C07163=1015.191,-31.274,-116.059,-24.116,21.567,-43.277
C07164=1015.192,-30.876,-116.091,-24.117,21.566,-43.271
C07165=1015.193,-30.478,-116.124,-24.117,21.565,-43.265
C07166=1015.195,-30.081,-116.155,-24.118,21.565,-43.260
C07167=1015.196,-29.684,-116.187,-24.119,21.565,-43.255
C07168=1015.197,-29.286,-116.220,-24.120,21.564,-43.249
C07169=1015.197,-28.889,-116.253,-24.120,21.563,-43.243
C07170=1015.198,-28.491,-116.285,-24.121,21.562,-43.238
C07171=1015.198,-28.094,-116.317,-24.122,21.562,-43.232
C07172=1015.200,-27.696,-116.350,-24.123,21.562,-43.227
C07173=1015.201,-27.299,-116.382,-24.123,21.561,-43.221
C07174=1015.201,-26.902,-116.414,-24.124,21.560,-43.217
C07175=1015.203,-26.504,-116.447,-24.125,21.560,-43.212
C07176=1015.203,-26.106,-116.479,-24.125,21.559,-43.206
C07177=1015.204,-25.709,-116.512,-24.126,21.558,-43.201
C07178=1015.205,-25.311,-116.544,-24.127,21.558,-43.195
C07179=1015.206,-24.914,-116.576,-24.128,21.558,-43.190
C07180=1015.206,-24.517,-116.610,-24.128,21.557,-43.184
C07181=1015.207,-24.120,-116.642,-24.129,21.556,-43.178
C07182=1015.207,-23.721,-116.675,-24.130,21.556,-43.173
C07183=1015.208,-23.324,-116.707,-24.131,21.555,-43.168
C07184=1015.209,-22.927,-116.740,-24.131,21.555,-43.162
C07185=1015.209,-22.529,-116.772,-24.132,21.554,-43.156
C07186=1015.210,-22.131,-116.805,-24.133,21.554,-43.151
C07187=1015.210,-21.734,-116.838,-24.134,21.553,-43.146
C07188=1015.210,-21.336,-116.870,-24.134,21.552,-43.140
C07189=1015.211,-20.939,-116.903,-24.135,21.553,-43.135
C07190=1015.212,-20.541,-116.936,-24.136,21.552,-43.129
C07191=1015.213,-20.144,-116.969,-24.136,21.551,-43.123
C07192=1015.213,-19.733,-117.002,-24.138,21.551,-43.116
C07193=1015.213,-19.483,-117.023,-24.138,21.550,-43.113
C07194=1015.213,-19.196,-117.047,-24.139,21.550,-43.109
C07195=1015.214,-18.884,-117.073,-24.139,21.550,-43.107
C07196=1015.215,-18.573,-117.098,-24.139,21.549,-43.105
C07197=1015.214,-18.285,-117.121,-24.139,21.549,-43.101
C07198=1015.214,-18.036,-117.142,-24.140,21.548,-43.098
C07199=1015.215,-17.626,-117.176,-24.141,21.547,-43.090
C07200=1015.215,-17.228,-117.209,-24.142,21.548,-43.085
C07201=1015.215,-16.831,-117.242,-24.142,21.547,-43.079
C07202=1015.216,-16.432,-117.274,-24.143,21.546,-43.074
C07203=1015.216,-16.032,-117.308,-24.144,21.546,-43.068
C07204=1015.217,-15.631,-117.341,-24.145,21.545,-43.063
C07205=1015.217,-15.228,-117.375,-24.145,21.545,-43.057
C07206=1015.216,-14.822,-117.408,-24.146,21.544,-43.052
C07207=1015.216,-14.414,-117.442,-24.147,21.544,-43.046
C07208=1015.217,-14.003,-117.476,-24.148,21.543,-43.041
C07209=1015.217,-13.588,-117.510,-24.148,21.543,-43.035
C07210=1015.217,-13.171,-117.545,-24.149,21.542,-43.029
C07211=1015.217,-12.751,-117.580,-24.150,21.542,-43.024
C07212=1015.217,-12.540,-117.598,-24.150,21.541,-43.022
C07213=1015.217,-12.329,-117.615,-24.151,21.541,-43.019
C07214=1015.217,-12.117,-117.633,-24.151,21.540,-43.016
C07215=1015.217,-11.905,-117.650,-24.151,21.540,-43.013
C07216=1015.217,-11.692,-117.668,-24.152,21.540,-43.011
C07217=1015.217,-11.479,-117.686,-24.152,21.540,-43.007
C07218=1015.217,-11.265,-117.704,-24.152,21.539,-43.006
C07219=1015.217,-11.051,-117.722,-24.153,21.539,-43.002
C07220=1015.216,-10.836,-117.740,-24.153,21.539,-42.998
C07221=1015.217,-10.621,-117.758,-24.154,21.538,-42.996
C07222=1015.216,-10.406,-117.776,-24.154,21.539,-42.993
C07223=1015.217,-10.189,-117.794,-24.154,21.538,-42.991
C07224=1015.217,-9.974,-117.811,-24.155,21.538,-42.987
C07225=1015.217,-9.758,-117.829,-24.155,21.538,-42.985
C07226=1015.216,-9.541,-117.848,-24.156,21.537,-42.982
C07227=1015.216,-9.325,-117.865,-24.156,21.537,-42.980
C07228=1015.216,-9.109,-117.883,-24.156,21.536,-42.976
C07229=1015.217,-8.892,-117.902,-24.157,21.537,-42.973
C07230=1015.217,-8.675,-117.920,-24.157,21.536,-42.971
C07231=1015.216,-8.459,-117.938,-24.158,21.536,-42.967
C07232=1015.216,-8.242,-117.956,-24.158,21.536,-42.965
C07233=1015.216,-8.026,-117.974,-24.158,21.535,-42.961
C07234=1015.216,-7.807,-117.992,-24.159,21.535,-42.959
C07235=1015.216,-7.588,-118.011,-24.159,21.534,-42.956
C07236=1015.216,-7.368,-118.029,-24.160,21.535,-42.952
C07237=1015.216,-7.146,-118.048,-24.160,21.534,-42.950
C07238=1015.216,-6.924,-118.067,-24.160,21.534,-42.947
C07239=1015.215,-6.701,-118.085,-24.161,21.533,-42.944
C07240=1015.216,-6.476,-118.104,-24.161,21.533,-42.941
C07241=1015.215,-6.252,-118.122,-24.161,21.533,-42.939
C07242=1015.215,-6.028,-118.142,-24.162,21.533,-42.935
C07243=1015.215,-5.804,-118.160,-24.162,21.532,-42.934
C07244=1015.215,-5.580,-118.179,-24.163,21.532,-42.930
C07245=1015.214,-5.357,-118.198,-24.163,21.532,-42.927
C07246=1015.214,-5.136,-118.216,-24.163,21.532,-42.925
C07247=1015.214,-4.917,-118.234,-24.164,21.531,-42.921
C07248=1015.213,-4.698,-118.253,-24.164,21.531,-42.919
C07249=1015.213,-4.481,-118.271,-24.165,21.531,-42.915
C07250=1015.213,-4.266,-118.290,-24.165,21.530,-42.913
C07251=1015.213,-4.052,-118.307,-24.165,21.530,-42.910
C07252=1015.213,-3.840,-118.325,-24.166,21.530,-42.908
C07253=1015.213,-3.629,-118.343,-24.166,21.530,-42.904
C07254=1015.212,-3.208,-118.379,-24.167,21.529,-42.899
C07255=1015.211,-2.788,-118.414,-24.168,21.529,-42.893
C07256=1015.211,-2.371,-118.449,-24.169,21.529,-42.888
C07257=1015.210,-1.955,-118.484,-24.169,21.528,-42.882
C07258=1015.210,-1.543,-118.518,-24.170,21.527,-42.877
C07259=1015.209,-1.133,-118.553,-24.171,21.527,-42.872
C07260=1015.209,-0.725,-118.588,-24.171,21.526,-42.867
C07261=1015.209,-0.320,-118.622,-24.172,21.525,-42.862
C07262=1015.208,0.084,-118.656,-24.173,21.525,-42.857
C07263=1015.207,0.486,-118.690,-24.173,21.525,-42.851
C07264=1015.206,0.885,-118.724,-24.174,21.525,-42.846
C07265=1015.206,1.284,-118.758,-24.175,21.523,-42.841
C07266=1015.206,1.682,-118.791,-24.175,21.524,-42.836
C07267=1015.205,2.068,-118.824,-24.176,21.523,-42.833
C07268=1015.203,2.420,-118.854,-24.177,21.522,-42.827
C07269=1015.203,2.744,-118.881,-24.177,21.522,-42.823
C07270=1015.203,3.056,-118.907,-24.178,21.521,-42.817
C07271=1015.202,3.384,-118.935,-24.179,21.521,-42.812
C07272=1015.202,3.744,-118.966,-24.179,21.521,-42.809
C07273=1015.200,4.133,-118.999,-24.180,21.520,-42.805
C07274=1015.199,4.529,-119.032,-24.180,21.519,-42.799
C07275=1015.199,4.924,-119.066,-24.181,21.520,-42.794
C07276=1015.198,5.319,-119.100,-24.182,21.519,-42.790
C07277=1015.197,5.714,-119.133,-24.182,21.518,-42.785
C07278=1015.196,6.108,-119.167,-24.183,21.519,-42.779
C07279=1015.195,6.500,-119.200,-24.184,21.517,-42.775
C07280=1015.194,6.893,-119.233,-24.185,21.517,-42.770
C07281=1015.193,7.284,-119.267,-24.185,21.517,-42.764
C07282=1015.193,7.671,-119.300,-24.186,21.516,-42.761
C07283=1015.191,8.055,-119.333,-24.187,21.516,-42.755
C07284=1015.190,8.436,-119.365,-24.187,21.515,-42.751
C07285=1015.190,8.815,-119.397,-24.188,21.515,-42.746
C07286=1015.189,9.191,-119.430,-24.189,21.514,-42.740
C07287=1015.187,9.566,-119.462,-24.189,21.514,-42.737
C07288=1015.186,9.943,-119.493,-24.190,21.513,-42.731
C07289=1015.185,10.321,-119.526,-24.191,21.513,-42.726
C07290=1015.184,10.702,-119.559,-24.191,21.513,-42.722
C07291=1015.183,11.085,-119.591,-24.192,21.512,-42.716
C07292=1015.182,11.470,-119.625,-24.192,21.511,-42.713
C07293=1015.181,11.856,-119.657,-24.193,21.512,-42.707
C07294=1015.179,12.244,-119.690,-24.193,21.510,-42.703
C07295=1015.178,12.630,-119.723,-24.194,21.510,-42.698
C07296=1015.177,13.016,-119.757,-24.195,21.511,-42.693
C07297=1015.176,13.403,-119.790,-24.196,21.509,-42.689
C07298=1015.175,13.791,-119.823,-24.196,21.509,-42.683
C07299=1015.173,14.178,-119.856,-24.197,21.509,-42.680
C07300=1015.172,14.566,-119.890,-24.198,21.508,-42.674
C07301=1015.171,14.955,-119.924,-24.198,21.508,-42.670
C07302=1015.169,15.345,-119.957,-24.199,21.507,-42.665
C07303=1015.168,15.735,-119.990,-24.200,21.507,-42.659
C07304=1015.166,16.126,-120.024,-24.200,21.506,-42.656
C07305=1015.165,16.517,-120.058,-24.201,21.506,-42.650
C07306=1015.163,16.910,-120.092,-24.201,21.505,-42.646
C07307=1015.162,17.304,-120.126,-24.202,21.505,-42.641
C07308=1015.161,17.698,-120.159,-24.203,21.505,-42.635
C07309=1015.159,18.094,-120.193,-24.203,21.504,-42.632
C07310=1015.158,18.489,-120.227,-24.204,21.503,-42.626
C07311=1015.156,18.886,-120.262,-24.205,21.503,-42.622
C07312=1015.155,19.282,-120.296,-24.205,21.503,-42.617
C07313=1015.154,19.493,-120.314,-24.206,21.503,-42.613
C07314=1015.153,19.730,-120.334,-24.206,21.502,-42.610
C07315=1015.151,19.995,-120.358,-24.207,21.503,-42.606
C07316=1015.151,20.282,-120.382,-24.207,21.501,-42.604
C07317=1015.149,20.579,-120.408,-24.207,21.501,-42.602
C07318=1015.148,20.871,-120.434,-24.208,21.502,-42.599
C07319=1015.147,21.143,-120.457,-24.208,21.501,-42.597
C07320=1015.146,21.387,-120.478,-24.209,21.501,-42.593
C07321=1015.145,21.802,-120.514,-24.210,21.501,-42.586
C07322=1015.143,22.176,-120.546,-24.210,21.500,-42.584
C07323=1015.142,22.498,-120.574,-24.211,21.500,-42.580
C07324=1015.140,22.764,-120.598,-24.211,21.500,-42.577
C07325=1015.139,22.996,-120.617,-24.211,21.499,-42.573
C07326=1015.138,23.230,-120.637,-24.212,21.498,-42.567
C07327=1015.137,23.502,-120.661,-24.213,21.498,-42.564
C07328=1015.135,23.832,-120.690,-24.213,21.498,-42.562
C07329=1015.134,24.215,-120.723,-24.213,21.497,-42.558
C07330=1015.132,24.614,-120.758,-24.214,21.497,-42.553
C07331=1015.130,25.014,-120.792,-24.215,21.497,-42.549
C07332=1015.129,25.413,-120.827,-24.215,21.496,-42.543
C07333=1015.126,25.812,-120.862,-24.216,21.496,-42.540
C07334=1015.124,26.212,-120.897,-24.217,21.496,-42.534
C07335=1015.122,26.611,-120.932,-24.218,21.495,-42.529
C07336=1015.121,27.010,-120.966,-24.218,21.494,-42.525
C07337=1015.119,27.410,-121.001,-24.219,21.495,-42.520
C07338=1015.116,27.809,-121.035,-24.219,21.493,-42.516
C07339=1015.114,28.208,-121.071,-24.220,21.493,-42.510
C07340=1015.112,28.608,-121.105,-24.221,21.493,-42.507
C07341=1015.110,29.008,-121.141,-24.221,21.492,-42.501
C07342=1015.108,29.408,-121.175,-24.222,21.492,-42.497
C07343=1015.106,29.807,-121.210,-24.223,21.492,-42.492
C07344=1015.104,30.206,-121.245,-24.223,21.491,-42.488
C07345=1015.102,30.606,-121.279,-24.224,21.491,-42.483
C07346=1015.100,31.006,-121.315,-24.224,21.490,-42.479
C07347=1015.098,31.404,-121.350,-24.225,21.490,-42.474
C07348=1015.095,31.804,-121.384,-24.226,21.489,-42.469
C07349=1015.093,32.204,-121.420,-24.226,21.489,-42.464
C07350=1015.091,32.604,-121.454,-24.227,21.489,-42.461
C07351=1015.089,33.003,-121.490,-24.228,21.489,-42.455
C07352=1015.086,33.403,-121.524,-24.228,21.487,-42.451
C07353=1015.084,33.803,-121.559,-24.229,21.488,-42.446
C07354=1015.082,34.202,-121.595,-24.229,21.487,-42.442
C07355=1015.079,34.602,-121.630,-24.230,21.486,-42.437
C07356=1015.077,35.002,-121.665,-24.231,21.486,-42.433
C07357=1015.075,35.402,-121.699,-24.231,21.486,-42.428
C07358=1015.073,35.801,-121.735,-24.232,21.486,-42.424
C07359=1015.070,36.201,-121.770,-24.233,21.485,-42.418
C07360=1015.068,36.601,-121.805,-24.233,21.484,-42.414
C07361=1015.065,37.001,-121.840,-24.234,21.485,-42.409
C07362=1015.063,37.401,-121.876,-24.235,21.484,-42.405
C07363=1015.060,37.801,-121.910,-24.235,21.483,-42.400
C07364=1015.058,38.200,-121.946,-24.236,21.483,-42.396
C07365=1015.055,38.600,-121.981,-24.237,21.483,-42.391
C07366=1015.053,39.000,-122.016,-24.237,21.483,-42.387
C07367=1015.050,39.400,-122.051,-24.238,21.482,-42.383
C07368=1015.047,39.800,-122.087,-24.238,21.481,-42.378
C07369=1015.045,40.200,-122.122,-24.239,21.481,-42.374
C07370=1015.042,40.600,-122.158,-24.240,21.481,-42.369
C07371=1015.040,41.000,-122.192,-24.240,21.481,-42.365
C07372=1015.037,41.399,-122.228,-24.241,21.480,-42.359
C07373=1015.033,41.799,-122.263,-24.241,21.479,-42.356
C07374=1015.031,42.199,-122.298,-24.242,21.479,-42.352
C07375=1015.028,42.599,-122.333,-24.243,21.479,-42.347
C07376=1015.025,42.999,-122.369,-24.243,21.479,-42.343
C07377=1015.023,43.399,-122.404,-24.244,21.479,-42.338
C07378=1015.020,43.799,-122.439,-24.244,21.477,-42.333
C07379=1015.017,44.199,-122.475,-24.245,21.477,-42.330
C07380=1015.014,44.599,-122.510,-24.246,21.477,-42.325
C07381=1015.011,44.999,-122.546,-24.246,21.477,-42.321
C07382=1015.009,45.399,-122.581,-24.247,21.477,-42.316
C07383=1015.006,45.799,-122.617,-24.247,21.475,-42.311
C07384=1015.003,46.199,-122.652,-24.248,21.475,-42.308
C07385=1015.000,46.599,-122.688,-24.249,21.475,-42.302
C07386=1014.997,46.999,-122.723,-24.249,21.475,-42.299
C07387=1014.994,47.400,-122.758,-24.250,21.474,-42.295
C07388=1014.991,47.799,-122.794,-24.251,21.474,-42.290
C07389=1014.987,48.200,-122.830,-24.251,21.474,-42.286
C07390=1014.985,48.599,-122.865,-24.251,21.472,-42.282
C07391=1014.982,49.000,-122.901,-24.252,21.473,-42.277
C07392=1014.979,49.400,-122.937,-24.253,21.472,-42.273
C07393=1014.975,49.800,-122.972,-24.254,21.472,-42.268
C07394=1014.973,50.200,-123.007,-24.254,21.472,-42.264
C07395=1014.970,50.600,-123.043,-24.255,21.471,-42.260
C07396=1014.966,51.001,-123.078,-24.255,21.471,-42.255
C07397=1014.963,51.401,-123.115,-24.256,21.471,-42.251
C07398=1014.960,51.801,-123.150,-24.256,21.470,-42.247
C07399=1014.957,52.201,-123.186,-24.257,21.469,-42.243
C07400=1014.953,52.601,-123.221,-24.258,21.469,-42.238
C07401=1014.949,53.001,-123.257,-24.258,21.469,-42.234
C07402=1014.946,53.401,-123.293,-24.259,21.468,-42.230
C07403=1014.943,53.801,-123.328,-24.259,21.468,-42.225
C07404=1014.940,54.201,-123.364,-24.260,21.468,-42.221
C07405=1014.937,54.602,-123.400,-24.260,21.468,-42.218
C07406=1014.933,55.002,-123.435,-24.261,21.468,-42.212
C07407=1014.930,55.402,-123.471,-24.262,21.467,-42.209
C07408=1014.927,55.803,-123.506,-24.262,21.467,-42.205
C07409=1014.923,56.202,-123.542,-24.263,21.465,-42.201
C07410=1014.920,56.602,-123.578,-24.264,21.466,-42.196
C07411=1014.916,57.002,-123.614,-24.264,21.465,-42.192
C07412=1014.913,57.403,-123.650,-24.264,21.465,-42.188
C07413=1014.909,57.803,-123.685,-24.265,21.465,-42.183
C07414=1014.906,58.203,-123.721,-24.266,21.464,-42.179
C07415=1014.901,58.603,-123.757,-24.266,21.464,-42.175
C07416=1014.898,59.003,-123.793,-24.267,21.463,-42.172
C07417=1014.895,59.403,-123.828,-24.268,21.464,-42.166
C07418=1014.891,59.804,-123.865,-24.268,21.463,-42.163
C07419=1014.887,60.203,-123.900,-24.269,21.463,-42.159
C07420=1014.884,60.603,-123.936,-24.269,21.462,-42.155
C07421=1014.880,61.004,-123.972,-24.270,21.462,-42.150
C07422=1014.877,61.405,-124.008,-24.270,21.462,-42.146
C07423=1014.872,61.804,-124.044,-24.271,21.461,-42.142
C07424=1014.869,62.204,-124.079,-24.271,21.461,-42.139
C07425=1014.865,62.624,-124.118,-24.272,21.460,-42.133
C07426=1014.862,62.877,-124.140,-24.272,21.460,-42.131
C07427=1014.860,63.145,-124.164,-24.273,21.460,-42.129
C07428=1014.858,63.395,-124.187,-24.273,21.459,-42.127
C07429=1014.856,63.612,-124.205,-24.274,21.460,-42.124
C07430=1014.854,63.819,-124.224,-24.274,21.460,-42.122
C07431=1014.852,64.036,-124.244,-24.274,21.459,-42.120
C07432=1014.849,64.266,-124.265,-24.274,21.459,-42.116
C07433=1014.848,64.502,-124.286,-24.275,21.459,-42.115
C07434=1014.845,64.738,-124.307,-24.275,21.458,-42.113
C07435=1014.842,64.968,-124.328,-24.275,21.458,-42.111
C07436=1014.840,65.188,-124.348,-24.276,21.459,-42.108
C07437=1014.838,65.402,-124.367,-24.276,21.458,-42.106
C07438=1014.834,65.810,-124.404,-24.277,21.458,-42.102
C07439=1014.830,66.207,-124.440,-24.277,21.457,-42.098
C07440=1014.827,66.608,-124.475,-24.278,21.457,-42.094
C07441=1014.822,67.010,-124.511,-24.278,21.457,-42.089
C07442=1014.818,67.414,-124.548,-24.279,21.457,-42.085
C07443=1014.814,67.818,-124.584,-24.279,21.456,-42.082
C07444=1014.810,68.224,-124.621,-24.280,21.456,-42.078
C07445=1014.806,68.632,-124.658,-24.280,21.455,-42.074
C07446=1014.801,69.040,-124.694,-24.281,21.455,-42.069
C07447=1014.796,69.451,-124.731,-24.282,21.455,-42.065
C07448=1014.793,69.861,-124.769,-24.282,21.454,-42.061
C07449=1014.788,70.273,-124.806,-24.283,21.454,-42.058
C07450=1014.784,70.684,-124.842,-24.283,21.453,-42.054
C07451=1014.780,71.095,-124.880,-24.284,21.454,-42.049
C07452=1014.775,71.505,-124.917,-24.285,21.453,-42.045
C07453=1014.771,71.918,-124.953,-24.285,21.453,-42.041
C07454=1014.767,72.332,-124.991,-24.285,21.452,-42.037
C07455=1014.762,72.746,-125.028,-24.286,21.452,-42.034
C07456=1014.758,73.164,-125.067,-24.287,21.452,-42.028
C07457=1014.753,73.584,-125.105,-24.287,21.452,-42.025
C07458=1014.751,73.796,-125.123,-24.288,21.451,-42.023
C07459=1014.749,74.008,-125.142,-24.288,21.451,-42.021
C07460=1014.746,74.221,-125.162,-24.288,21.451,-42.019
C07461=1014.744,74.434,-125.181,-24.288,21.451,-42.017
C07462=1014.741,74.647,-125.200,-24.289,21.450,-42.015
C07463=1014.738,74.861,-125.220,-24.289,21.451,-42.012
C07464=1014.736,75.074,-125.239,-24.289,21.451,-42.010
C07465=1014.734,75.286,-125.258,-24.290,21.450,-42.008
C07466=1014.729,75.706,-125.296,-24.290,21.450,-42.004
C07467=1014.724,76.118,-125.333,-24.291,21.449,-42.001
C07468=1014.719,76.520,-125.370,-24.291,21.449,-41.997
C07469=1014.715,76.915,-125.405,-24.292,21.449,-41.994
C07470=1014.711,77.303,-125.441,-24.292,21.448,-41.989
C07471=1014.707,77.689,-125.476,-24.293,21.447,-41.986
C07472=1014.702,78.075,-125.511,-24.293,21.448,-41.980
C07473=1014.698,78.465,-125.546,-24.294,21.447,-41.977
C07474=1014.692,78.863,-125.582,-24.294,21.447,-41.973
C07475=1014.688,79.268,-125.618,-24.295,21.447,-41.970
C07476=1014.683,79.683,-125.656,-24.296,21.447,-41.966
C07477=1014.681,79.893,-125.675,-24.296,21.446,-41.964
C07478=1014.678,80.104,-125.694,-24.296,21.446,-41.962
C07479=1014.675,80.317,-125.713,-24.296,21.446,-41.960
C07480=1014.673,80.530,-125.733,-24.297,21.446,-41.958
C07481=1014.670,80.743,-125.752,-24.297,21.445,-41.956
C07482=1014.668,80.955,-125.772,-24.297,21.445,-41.955
C07483=1014.665,81.168,-125.791,-24.297,21.445,-41.953
C07484=1014.663,81.380,-125.810,-24.298,21.445,-41.951
C07485=1014.660,81.593,-125.829,-24.298,21.445,-41.949
C07486=1014.657,81.804,-125.848,-24.298,21.444,-41.947
C07487=1014.655,82.016,-125.867,-24.299,21.445,-41.944
C07488=1014.652,82.227,-125.887,-24.299,21.444,-41.942
C07489=1014.647,82.647,-125.924,-24.299,21.444,-41.938
C07490=1014.641,83.068,-125.963,-24.300,21.444,-41.935
C07491=1014.637,83.486,-126.001,-24.300,21.444,-41.931
C07492=1014.632,83.904,-126.039,-24.301,21.443,-41.927
C07493=1014.626,84.320,-126.077,-24.301,21.443,-41.923
C07494=1014.621,84.734,-126.115,-24.302,21.443,-41.920
C07495=1014.616,85.146,-126.151,-24.302,21.442,-41.916
C07496=1014.611,85.557,-126.189,-24.303,21.442,-41.912
C07497=1014.605,85.965,-126.226,-24.303,21.441,-41.908
C07498=1014.601,86.373,-126.263,-24.304,21.442,-41.905
C07499=1014.595,86.779,-126.300,-24.304,21.441,-41.901
C07500=1014.590,87.182,-126.336,-24.305,21.441,-41.898
C07501=1014.584,87.578,-126.373,-24.305,21.440,-41.894
C07502=1014.579,87.966,-126.408,-24.306,21.440,-41.890
C07503=1014.575,88.349,-126.443,-24.307,21.440,-41.887
C07504=1014.570,88.732,-126.477,-24.307,21.440,-41.883
C07505=1014.565,89.118,-126.513,-24.308,21.439,-41.879
C07506=1014.559,89.510,-126.548,-24.308,21.439,-41.875
C07507=1014.554,89.910,-126.585,-24.309,21.439,-41.872
C07508=1014.549,90.308,-126.621,-24.309,21.439,-41.868
C07509=1014.543,90.707,-126.658,-24.310,21.438,-41.865
C07510=1014.538,91.106,-126.693,-24.310,21.438,-41.861
C07511=1014.532,91.505,-126.730,-24.311,21.438,-41.857
C07512=1014.526,91.904,-126.767,-24.311,21.438,-41.854
C07513=1014.521,92.303,-126.803,-24.312,21.437,-41.850
C07514=1014.516,92.702,-126.839,-24.312,21.437,-41.846
C07515=1014.510,93.102,-126.875,-24.312,21.437,-41.844
C07516=1014.505,93.500,-126.911,-24.313,21.436,-41.841
C07517=1014.499,93.899,-126.948,-24.313,21.436,-41.837
C07518=1014.493,94.298,-126.984,-24.314,21.435,-41.833
C07519=1014.488,94.697,-127.020,-24.315,21.436,-41.830
C07520=1014.482,95.096,-127.057,-24.315,21.435,-41.826
C07521=1014.476,95.495,-127.093,-24.316,21.435,-41.822
C07522=1014.470,95.894,-127.130,-24.316,21.435,-41.819
C07523=1014.465,96.293,-127.166,-24.317,21.435,-41.815
C07524=1014.460,96.691,-127.202,-24.317,21.434,-41.811
C07525=1014.453,97.090,-127.238,-24.318,21.434,-41.808
C07526=1014.447,97.489,-127.275,-24.318,21.433,-41.806
C07527=1014.442,97.888,-127.311,-24.318,21.433,-41.802
C07528=1014.435,98.286,-127.348,-24.319,21.432,-41.798
C07529=1014.430,98.685,-127.384,-24.319,21.433,-41.795
C07530=1014.423,99.084,-127.420,-24.320,21.432,-41.791
C07531=1014.418,99.482,-127.456,-24.320,21.432,-41.787
C07532=1014.413,99.881,-127.493,-24.321,21.432,-41.784
C07533=1014.406,100.280,-127.529,-24.322,21.432,-41.780
C07534=1014.400,100.678,-127.565,-24.322,21.431,-41.778
C07535=1014.394,101.077,-127.602,-24.322,21.431,-41.775
C07536=1014.388,101.476,-127.638,-24.323,21.431,-41.771
C07537=1014.382,101.875,-127.675,-24.323,21.430,-41.767
C07538=1014.376,102.273,-127.711,-24.324,21.430,-41.763
C07539=1014.369,102.671,-127.747,-24.324,21.430,-41.760
C07540=1014.363,103.071,-127.784,-24.325,21.430,-41.756
C07541=1014.357,103.469,-127.821,-24.325,21.430,-41.754
C07542=1014.350,103.867,-127.857,-24.326,21.429,-41.751
C07543=1014.344,104.266,-127.893,-24.326,21.429,-41.747
C07544=1014.338,104.665,-127.930,-24.327,21.429,-41.743
C07545=1014.332,105.063,-127.966,-24.327,21.429,-41.740
C07546=1014.325,105.461,-128.002,-24.328,21.428,-41.736
C07547=1014.319,105.860,-128.038,-24.328,21.428,-41.734
C07548=1014.313,106.259,-128.075,-24.328,21.427,-41.730
C07549=1014.306,106.658,-128.112,-24.329,21.427,-41.727
C07550=1014.300,107.056,-128.148,-24.330,21.427,-41.723
C07551=1014.294,107.454,-128.184,-24.330,21.427,-41.719
C07552=1014.286,107.853,-128.221,-24.330,21.426,-41.717
C07553=1014.280,108.251,-128.257,-24.331,21.426,-41.714
C07554=1014.274,108.650,-128.293,-24.331,21.426,-41.710
C07555=1014.267,109.048,-128.330,-24.332,21.426,-41.707
C07556=1014.260,109.447,-128.366,-24.332,21.426,-41.703
C07557=1014.254,109.845,-128.402,-24.333,21.425,-41.701
C07558=1014.247,110.244,-128.439,-24.333,21.425,-41.697
C07559=1014.241,110.642,-128.475,-24.334,21.425,-41.694
C07560=1014.233,111.040,-128.512,-24.334,21.425,-41.690
C07561=1014.227,111.438,-128.548,-24.334,21.424,-41.688
C07562=1014.220,111.837,-128.585,-24.335,21.423,-41.684
C07563=1014.213,112.235,-128.621,-24.335,21.424,-41.681
C07564=1014.206,112.634,-128.658,-24.336,21.423,-41.677
C07565=1014.199,113.031,-128.694,-24.336,21.423,-41.675
C07566=1014.192,113.430,-128.731,-24.337,21.423,-41.671
C07567=1014.186,113.828,-128.767,-24.337,21.422,-41.668
C07568=1014.178,114.228,-128.803,-24.338,21.423,-41.664
C07569=1014.171,114.625,-128.839,-24.338,21.422,-41.662
C07570=1014.164,115.024,-128.876,-24.339,21.422,-41.659
C07571=1014.157,115.422,-128.912,-24.339,21.422,-41.655
C07572=1014.150,115.820,-128.948,-24.340,21.422,-41.652
C07573=1014.143,116.219,-128.985,-24.340,21.421,-41.649
C07574=1014.136,116.617,-129.021,-24.340,21.420,-41.646
C07575=1014.128,117.016,-129.058,-24.341,21.421,-41.642
C07576=1014.121,117.414,-129.093,-24.341,21.420,-41.638
C07577=1014.114,117.813,-129.130,-24.342,21.420,-41.637
C07578=1014.106,118.210,-129.167,-24.342,21.420,-41.633
C07579=1014.099,118.609,-129.203,-24.343,21.420,-41.629
C07580=1014.092,119.007,-129.240,-24.343,21.420,-41.626
C07581=1014.085,119.406,-129.275,-24.343,21.419,-41.624
C07582=1014.077,119.804,-129.312,-24.344,21.419,-41.620
C07583=1014.070,120.202,-129.348,-24.345,21.419,-41.617
C07584=1014.063,120.601,-129.385,-24.345,21.418,-41.614
C07585=1014.056,120.999,-129.422,-24.345,21.418,-41.611
C07586=1014.048,121.397,-129.458,-24.346,21.418,-41.607
C07587=1014.042,121.796,-129.494,-24.346,21.417,-41.605
C07588=1014.034,122.194,-129.531,-24.347,21.418,-41.602
C07589=1014.027,122.593,-129.568,-24.347,21.417,-41.598
C07590=1014.020,122.991,-129.605,-24.348,21.418,-41.595
C07591=1014.013,123.389,-129.641,-24.348,21.416,-41.592
C07592=1014.006,123.788,-129.678,-24.348,21.417,-41.589
C07593=1013.998,124.187,-129.715,-24.349,21.416,-41.585
C07594=1013.991,124.585,-129.751,-24.349,21.416,-41.583
C07595=1013.984,124.983,-129.788,-24.350,21.416,-41.580
C07596=1013.976,125.381,-129.825,-24.350,21.416,-41.576
C07597=1013.969,125.780,-129.861,-24.350,21.415,-41.574
C07598=1013.962,126.179,-129.898,-24.351,21.415,-41.571
C07599=1013.954,126.577,-129.935,-24.351,21.415,-41.567
C07600=1013.947,126.975,-129.971,-24.352,21.415,-41.565
C07601=1013.939,127.373,-130.008,-24.352,21.414,-41.561
C07602=1013.932,127.772,-130.045,-24.353,21.415,-41.558
C07603=1013.924,128.170,-130.082,-24.353,21.414,-41.555
C07604=1013.917,128.569,-130.119,-24.354,21.414,-41.552
C07605=1013.909,128.967,-130.155,-24.354,21.413,-41.550
C07606=1013.902,129.365,-130.192,-24.354,21.413,-41.547
C07607=1013.894,129.764,-130.228,-24.355,21.413,-41.543
C07608=1013.886,130.163,-130.265,-24.355,21.413,-41.541
C07609=1013.879,130.561,-130.301,-24.356,21.413,-41.538
C07610=1013.871,130.959,-130.338,-24.356,21.413,-41.534
C07611=1013.863,131.358,-130.375,-24.356,21.412,-41.532
C07612=1013.855,131.756,-130.411,-24.357,21.412,-41.528
C07613=1013.847,132.155,-130.448,-24.357,21.412,-41.525
C07614=1013.840,132.553,-130.485,-24.358,21.411,-41.523
C07615=1013.831,132.952,-130.522,-24.358,21.412,-41.519
C07616=1013.823,133.350,-130.558,-24.358,21.411,-41.517
C07617=1013.815,133.749,-130.595,-24.359,21.411,-41.514
C07618=1013.807,134.148,-130.631,-24.359,21.411,-41.510
C07619=1013.799,134.546,-130.668,-24.360,21.410,-41.508
C07620=1013.791,134.944,-130.704,-24.360,21.411,-41.505
C07621=1013.783,135.340,-130.741,-24.360,21.410,-41.502
C07622=1013.775,135.711,-130.774,-24.361,21.409,-41.500
C07623=1013.768,136.050,-130.806,-24.361,21.410,-41.497
C07624=1013.762,136.368,-130.835,-24.361,21.409,-41.495
C07625=1013.755,136.685,-130.864,-24.362,21.409,-41.491
C07626=1013.748,137.021,-130.895,-24.363,21.410,-41.488
C07627=1013.741,137.390,-130.928,-24.363,21.408,-41.486
C07628=1013.732,137.791,-130.965,-24.363,21.408,-41.484
C07629=1013.728,137.996,-130.984,-24.363,21.408,-41.482
C07630=1013.723,138.213,-131.004,-24.364,21.408,-41.480
C07631=1013.718,138.451,-131.026,-24.364,21.408,-41.478
C07632=1013.712,138.710,-131.050,-24.364,21.407,-41.476
C07633=1013.707,138.988,-131.075,-24.364,21.408,-41.475
C07634=1013.700,139.275,-131.101,-24.365,21.408,-41.473
C07635=1013.694,139.563,-131.128,-24.365,21.408,-41.471
C07636=1013.688,139.840,-131.153,-24.365,21.408,-41.470
C07637=1013.683,140.099,-131.177,-24.366,21.408,-41.468
C07638=1013.678,140.334,-131.199,-24.366,21.408,-41.466
C07639=1013.668,140.751,-131.236,-24.366,21.407,-41.462
C07640=1013.660,141.156,-131.273,-24.366,21.406,-41.460
C07641=1013.651,141.561,-131.311,-24.367,21.407,-41.457
C07642=1013.642,141.967,-131.348,-24.368,21.406,-41.453
C07643=1013.633,142.373,-131.386,-24.368,21.406,-41.451
C07644=1013.624,142.782,-131.423,-24.368,21.406,-41.448
C07645=1013.615,143.191,-131.460,-24.369,21.405,-41.445
C07646=1013.605,143.599,-131.497,-24.369,21.406,-41.442
C07647=1013.597,144.009,-131.534,-24.370,21.405,-41.438
C07648=1013.587,144.420,-131.572,-24.370,21.405,-41.436
C07649=1013.578,144.832,-131.610,-24.370,21.405,-41.432
C07650=1013.568,145.243,-131.648,-24.371,21.404,-41.431
C07651=1013.559,145.655,-131.685,-24.371,21.405,-41.427
C07652=1013.549,146.068,-131.723,-24.372,21.404,-41.424
C07653=1013.542,146.377,-131.751,-24.372,21.404,-41.422
C07654=1013.515,147.591,-131.861,-24.540,22.052,-41.028
C07655=1013.508,147.860,-131.887,-24.577,22.199,-40.939
C07656=1013.502,148.138,-131.912,-24.616,22.351,-40.849
C07657=1013.494,148.423,-131.937,-24.654,22.506,-40.757
C07658=1013.488,148.714,-131.963,-24.694,22.666,-40.663
C07659=1013.481,149.010,-131.991,-24.734,22.828,-40.570
C07660=1013.474,149.309,-132.018,-24.774,22.993,-40.474
C07661=1013.467,149.610,-132.045,-24.814,23.158,-40.379
C07662=1013.460,149.909,-132.073,-24.853,23.322,-40.286
C07663=1013.454,150.206,-132.099,-24.892,23.487,-40.192
C07664=1013.447,150.497,-132.126,-24.930,23.649,-40.102
C07665=1013.440,150.783,-132.152,-24.967,23.807,-40.013
C07666=1013.433,151.062,-132.177,-25.003,23.962,-39.926
C07667=1013.427,151.333,-132.202,-25.038,24.113,-39.842
C07668=1013.421,151.596,-132.225,-25.071,24.258,-39.762
C07669=1013.415,151.850,-132.249,-25.103,24.400,-39.683
C07670=1013.409,152.099,-132.271,-25.135,24.540,-39.606
C07671=1013.404,152.343,-132.293,-25.165,24.676,-39.532
C07672=1013.398,152.585,-132.315,-25.195,24.812,-39.459
C07673=1013.392,152.826,-132.337,-25.225,24.947,-39.386
C07674=1013.387,153.067,-132.358,-25.255,25.083,-39.312
C07675=1013.381,153.308,-132.381,-25.284,25.219,-39.240
C07676=1013.375,153.550,-132.402,-25.314,25.356,-39.168
C07677=1013.370,153.791,-132.424,-25.343,25.491,-39.097
C07678=1013.365,154.032,-132.445,-25.372,25.627,-39.025
C07679=1013.359,154.272,-132.467,-25.401,25.764,-38.954
C07680=1013.353,154.513,-132.489,-25.429,25.900,-38.884
C07681=1013.348,154.753,-132.511,-25.458,26.037,-38.813
C07682=1013.342,154.992,-132.533,-25.486,26.173,-38.743
C07683=1013.337,155.232,-132.554,-25.514,26.310,-38.672
C07684=1013.331,155.472,-132.575,-25.542,26.447,-38.603
C07685=1013.326,155.711,-132.597,-25.569,26.583,-38.534
C07686=1013.320,155.950,-132.619,-25.597,26.719,-38.465
C07687=1013.315,156.190,-132.640,-25.624,26.857,-38.396
C07688=1013.310,156.429,-132.662,-25.652,26.994,-38.328
C07689=1013.303,156.668,-132.683,-25.679,27.132,-38.260
C07690=1013.295,157.070,-132.719,-25.724,27.362,-38.147
C07691=1013.287,157.384,-132.748,-25.759,27.544,-38.058
C07692=1013.282,157.622,-132.769,-25.785,27.680,-37.991
C07693=1013.276,157.859,-132.790,-25.811,27.817,-37.925
C07694=1013.271,158.096,-132.811,-25.837,27.955,-37.859
C07695=1013.265,158.331,-132.832,-25.862,28.091,-37.795
C07696=1013.260,158.566,-132.854,-25.888,28.227,-37.729
C07697=1013.254,158.801,-132.875,-25.913,28.364,-37.665
C07698=1013.249,159.037,-132.896,-25.938,28.501,-37.599
C07699=1013.243,159.273,-132.916,-25.963,28.638,-37.536
C07700=1013.239,159.507,-132.938,-25.988,28.775,-37.472
C07701=1013.232,159.739,-132.958,-26.012,28.910,-37.409
C07702=1013.230,159.972,-132.981,-26.026,28.985,-37.375
C07703=1013.229,160.206,-133.005,-26.028,28.996,-37.368
C07704=1013.228,160.445,-133.030,-26.030,29.007,-37.362
C07705=1013.227,160.696,-133.056,-26.032,29.019,-37.354
C07706=1013.226,160.958,-133.083,-26.034,29.031,-37.348
C07707=1013.224,161.235,-133.112,-26.037,29.045,-37.339
C07708=1013.223,161.528,-133.143,-26.039,29.058,-37.332
C07709=1013.221,161.831,-133.174,-26.042,29.072,-37.323
C07710=1013.220,162.137,-133.206,-26.044,29.085,-37.316
C07711=1013.218,162.429,-133.236,-26.047,29.099,-37.308
C07712=1013.217,162.736,-133.269,-26.049,29.113,-37.301
C07713=1013.216,163.030,-133.299,-26.052,29.126,-37.292
C07714=1013.215,163.293,-133.326,-26.054,29.138,-37.286
C07715=1013.213,163.531,-133.351,-26.056,29.148,-37.279
C07716=1013.212,163.751,-133.374,-26.058,29.158,-37.274
C07717=1013.211,164.086,-133.409,-26.061,29.175,-37.265
C07718=1013.210,164.360,-133.438,-26.063,29.187,-37.257
C07719=1013.209,164.678,-133.471,-26.066,29.201,-37.251
C07720=1013.207,164.981,-133.503,-26.068,29.215,-37.242
C07721=1013.206,165.216,-133.527,-26.070,29.225,-37.235
C07722=1013.206,165.451,-133.551,-26.073,29.237,-37.229
C07723=1013.204,165.687,-133.576,-26.074,29.247,-37.224
C07724=1013.203,165.923,-133.601,-26.076,29.257,-37.217
C07725=1013.202,166.158,-133.625,-26.078,29.267,-37.211
C07726=1013.202,166.393,-133.650,-26.080,29.279,-37.205
C07727=1013.201,166.629,-133.675,-26.082,29.289,-37.198
C07728=1013.199,166.864,-133.699,-26.084,29.300,-37.193
C07729=1013.198,167.100,-133.724,-26.086,29.311,-37.187
C07730=1013.197,167.335,-133.748,-26.088,29.322,-37.180
C07731=1013.196,167.571,-133.773,-26.090,29.334,-37.174
C07732=1013.195,167.806,-133.798,-26.093,29.346,-37.166
C07733=1013.194,168.042,-133.823,-26.094,29.356,-37.161
C07734=1013.193,168.278,-133.847,-26.097,29.367,-37.155
C07735=1013.193,168.513,-133.872,-26.098,29.377,-37.149
C07736=1013.191,168.749,-133.896,-26.100,29.388,-37.143
C07737=1013.190,168.984,-133.921,-26.102,29.399,-37.136
C07738=1013.189,169.220,-133.946,-26.104,29.411,-37.130
C07739=1013.189,169.455,-133.970,-26.106,29.420,-37.125
C07740=1013.187,169.690,-133.995,-26.109,29.433,-37.117
C07741=1013.186,169.926,-134.020,-26.111,29.444,-37.111
C07742=1013.185,170.162,-134.045,-26.113,29.457,-37.105
C07743=1013.184,170.398,-134.070,-26.115,29.467,-37.098
C07744=1013.183,170.633,-134.095,-26.117,29.477,-37.093
C07745=1013.183,170.868,-134.119,-26.119,29.488,-37.086
C07746=1013.181,171.104,-134.144,-26.120,29.498,-37.081
C07747=1013.180,171.340,-134.169,-26.122,29.510,-37.075
C07748=1013.179,171.575,-134.193,-26.124,29.520,-37.068
C07749=1013.179,171.811,-134.218,-26.126,29.532,-37.062
C07750=1013.178,172.047,-134.242,-26.129,29.543,-37.056
C07751=1013.177,172.282,-134.267,-26.131,29.557,-37.049
C07752=1013.176,172.517,-134.292,-26.133,29.568,-37.042
C07753=1013.174,172.753,-134.317,-26.135,29.578,-37.037
C07754=1013.174,172.989,-134.342,-26.137,29.588,-37.030
C07755=1013.173,173.225,-134.367,-26.139,29.599,-37.025
C07756=1013.171,173.460,-134.392,-26.141,29.610,-37.019
C07757=1013.171,173.695,-134.416,-26.143,29.621,-37.012
C07758=1013.170,173.932,-134.441,-26.145,29.633,-37.006
C07759=1013.169,174.167,-134.466,-26.147,29.644,-37.000
C07760=1013.168,174.402,-134.491,-26.149,29.657,-36.992
C07761=1013.167,174.638,-134.516,-26.151,29.669,-36.986
C07762=1013.166,174.874,-134.541,-26.153,29.680,-36.980
C07763=1013.165,175.110,-134.565,-26.155,29.690,-36.975
C07764=1013.164,175.345,-134.590,-26.157,29.702,-36.969
C07765=1013.163,175.581,-134.616,-26.159,29.712,-36.962
C07766=1013.163,175.817,-134.640,-26.161,29.724,-36.956
C07767=1013.162,176.052,-134.665,-26.163,29.735,-36.949
C07768=1013.161,176.288,-134.690,-26.165,29.747,-36.943
C07769=1013.160,176.524,-134.715,-26.167,29.758,-36.937
C07770=1013.159,176.759,-134.740,-26.169,29.770,-36.931
C07771=1013.158,176.995,-134.765,-26.171,29.782,-36.925
C07772=1013.156,177.231,-134.789,-26.174,29.795,-36.917
C07773=1013.156,177.466,-134.815,-26.175,29.804,-36.912
C07774=1013.155,177.702,-134.840,-26.177,29.816,-36.906
C07775=1013.154,177.938,-134.864,-26.179,29.827,-36.899
C07776=1013.153,178.174,-134.890,-26.181,29.837,-36.894
C07777=1013.152,178.409,-134.915,-26.183,29.849,-36.888
C07778=1013.152,178.645,-134.939,-26.185,29.861,-36.880
C07779=1013.151,178.880,-134.964,-26.187,29.873,-36.874
C07780=1013.150,179.116,-134.989,-26.189,29.885,-36.868
C07781=1013.149,179.352,-135.014,-26.192,29.897,-36.861
C07782=1013.148,179.587,-135.039,-26.194,29.909,-36.854
C07783=1013.147,179.823,-135.064,-26.196,29.920,-36.850
C07784=1013.146,180.059,-135.089,-26.198,29.931,-36.843
C07785=1013.145,180.295,-135.114,-26.200,29.942,-36.837
C07786=1013.144,180.531,-135.139,-26.202,29.953,-36.830
C07787=1013.143,180.766,-135.164,-26.204,29.965,-36.824
C07788=1013.142,181.002,-135.189,-26.206,29.976,-36.818
C07789=1013.141,181.238,-135.214,-26.208,29.989,-36.812
C07790=1013.140,181.473,-135.239,-26.210,30.001,-36.805
C07791=1013.140,181.710,-135.264,-26.212,30.013,-36.799
C07792=1013.138,181.945,-135.289,-26.214,30.025,-36.793
C07793=1013.138,182.181,-135.314,-26.216,30.035,-36.786
C07794=1013.137,182.416,-135.340,-26.218,30.046,-36.781
C07795=1013.136,182.653,-135.364,-26.220,30.058,-36.775
C07796=1013.135,182.888,-135.389,-26.222,30.069,-36.769
C07797=1013.135,183.124,-135.415,-26.224,30.081,-36.762
C07798=1013.133,183.359,-135.440,-26.226,30.094,-36.755
C07799=1013.133,183.596,-135.465,-26.228,30.105,-36.749
C07800=1013.132,183.831,-135.490,-26.230,30.119,-36.742
C07801=1013.131,184.067,-135.515,-26.232,30.130,-36.736
C07802=1013.130,184.302,-135.540,-26.234,30.142,-36.730
C07803=1013.130,184.538,-135.566,-26.236,30.153,-36.723
C07804=1013.128,184.774,-135.590,-26.238,30.164,-36.719
C07805=1013.128,185.010,-135.616,-26.240,30.175,-36.712
C07806=1013.127,185.245,-135.641,-26.242,30.187,-36.706
C07807=1013.126,185.481,-135.666,-26.244,30.199,-36.699
C07808=1013.125,185.717,-135.691,-26.246,30.212,-36.693
C07809=1013.124,185.953,-135.716,-26.248,30.223,-36.687
C07810=1013.123,186.188,-135.741,-26.251,30.236,-36.680
C07811=1013.123,186.424,-135.767,-26.253,30.249,-36.674
C07812=1013.122,186.660,-135.792,-26.255,30.260,-36.668
C07813=1013.121,186.895,-135.817,-26.257,30.271,-36.661
C07814=1013.120,187.132,-135.842,-26.259,30.282,-36.655
C07815=1013.119,187.367,-135.867,-26.261,30.294,-36.649
C07816=1013.119,187.603,-135.892,-26.263,30.306,-36.643
C07817=1013.118,187.839,-135.917,-26.265,30.318,-36.637
C07818=1013.117,188.075,-135.943,-26.267,30.330,-36.631
C07819=1013.116,188.311,-135.969,-26.269,30.343,-36.623
C07820=1013.115,188.547,-135.993,-26.271,30.356,-36.616
C07821=1013.114,188.783,-136.019,-26.273,30.368,-36.611
C07822=1013.113,189.018,-136.044,-26.275,30.380,-36.604
C07823=1013.113,189.254,-136.069,-26.277,30.391,-36.598
C07824=1013.112,189.490,-136.095,-26.279,30.403,-36.592
C07825=1013.111,189.725,-136.120,-26.281,30.414,-36.586
C07826=1013.111,189.961,-136.145,-26.283,30.426,-36.580
C07827=1013.110,190.197,-136.171,-26.285,30.438,-36.574
C07828=1013.109,190.433,-136.195,-26.287,30.450,-36.568
C07829=1013.108,190.669,-136.221,-26.289,30.463,-36.561
C07830=1013.108,190.905,-136.246,-26.292,30.476,-36.554
C07831=1013.107,191.140,-136.271,-26.294,30.489,-36.548
C07832=1013.106,191.376,-136.297,-26.296,30.500,-36.542
C07833=1013.105,191.612,-136.323,-26.298,30.512,-36.536
C07834=1013.104,191.848,-136.348,-26.300,30.523,-36.529
C07835=1013.104,192.084,-136.373,-26.301,30.535,-36.523
C07836=1013.103,192.320,-136.399,-26.303,30.546,-36.517
C07837=1013.103,192.556,-136.424,-26.305,30.559,-36.511
C07838=1013.102,192.791,-136.449,-26.308,30.572,-36.504
C07839=1013.101,193.027,-136.475,-26.310,30.584,-36.499
C07840=1013.100,193.263,-136.499,-26.312,30.597,-36.492
C07841=1013.099,193.499,-136.525,-26.314,30.611,-36.485
C07842=1013.099,193.735,-136.550,-26.316,30.622,-36.478
C07843=1013.097,193.971,-136.576,-26.318,30.633,-36.474
C07844=1013.097,194.207,-136.602,-26.320,30.644,-36.467
C07845=1013.096,194.442,-136.627,-26.322,30.656,-36.461
C07846=1013.095,194.678,-136.652,-26.324,30.669,-36.454
C07847=1013.095,194.914,-136.678,-26.326,30.681,-36.448
C07848=1013.095,195.150,-136.703,-26.328,30.694,-36.441
C07849=1013.093,195.385,-136.728,-26.330,30.706,-36.435
C07850=1013.093,195.621,-136.754,-26.332,30.719,-36.428
C07851=1013.092,195.857,-136.780,-26.335,30.733,-36.421
C07852=1013.091,196.093,-136.805,-26.336,30.743,-36.416
C07853=1013.091,196.329,-136.831,-26.338,30.755,-36.410
C07854=1013.090,196.565,-136.856,-26.340,30.767,-36.405
C07855=1013.090,196.800,-136.882,-26.342,30.779,-36.398
C07856=1013.089,197.036,-136.907,-26.345,30.792,-36.391
C07857=1013.089,197.272,-136.933,-26.346,30.804,-36.385
C07858=1013.088,197.508,-136.958,-26.349,30.817,-36.378
C07859=1013.086,197.743,-136.984,-26.351,30.831,-36.372
C07860=1013.086,197.979,-137.009,-26.353,30.843,-36.366
C07861=1013.085,198.226,-137.036,-26.355,30.857,-36.358
C07862=1013.084,198.618,-137.078,-26.359,30.878,-36.348
C07863=1013.083,199.009,-137.121,-26.362,30.898,-36.339
C07864=1013.083,199.250,-137.147,-26.364,30.911,-36.332
C07865=1013.082,199.479,-137.172,-26.366,30.923,-36.326
C07866=1013.081,199.712,-137.197,-26.368,30.936,-36.319
C07867=1013.081,199.953,-137.223,-26.370,30.948,-36.313
C07868=1013.080,200.207,-137.250,-26.372,30.962,-36.306
C07869=1013.079,200.462,-137.279,-26.375,30.975,-36.299
C07870=1013.079,200.701,-137.304,-26.377,30.988,-36.292
C07871=1013.078,200.923,-137.329,-26.379,31.000,-36.286
C07872=1013.077,201.140,-137.352,-26.380,31.011,-36.282
C07873=1013.076,201.556,-137.397,-26.384,31.033,-36.271
C07874=1013.076,201.762,-137.420,-26.386,31.044,-36.264
C07875=1013.076,201.981,-137.443,-26.388,31.057,-36.258
C07876=1013.078,203.216,-137.580,-26.364,31.070,-36.698
C07877=1013.079,203.464,-137.607,-26.366,31.081,-36.692
C07878=1013.081,203.709,-137.634,-26.368,31.094,-36.686
C07879=1013.083,203.954,-137.660,-26.370,31.107,-36.681
C07880=1013.084,204.199,-137.687,-26.372,31.119,-36.675
C07881=1013.086,204.442,-137.714,-26.374,31.131,-36.670
C07882=1013.088,204.686,-137.740,-26.376,31.144,-36.664
C07883=1013.089,204.930,-137.767,-26.378,31.156,-36.658
C07884=1013.090,205.174,-137.794,-26.381,31.168,-36.653
C07885=1013.093,205.418,-137.821,-26.383,31.181,-36.647
C07886=1013.094,205.661,-137.848,-26.385,31.193,-36.642
C07887=1013.096,205.905,-137.874,-26.387,31.206,-36.636
C07888=1013.097,206.148,-137.900,-26.389,31.217,-36.630
C07889=1013.099,206.391,-137.927,-26.391,31.229,-36.624
C07890=1013.101,206.634,-137.954,-26.393,31.242,-36.619
C07891=1013.102,206.877,-137.981,-26.395,31.254,-36.613
C07892=1013.104,207.119,-138.007,-26.397,31.266,-36.607
C07893=1013.106,207.363,-138.033,-26.399,31.278,-36.601
C07894=1013.108,207.604,-138.060,-26.401,31.291,-36.596
C07895=1013.108,207.847,-138.087,-26.403,31.303,-36.590
C07896=1013.110,208.090,-138.113,-26.405,31.315,-36.584
C07897=1013.112,208.332,-138.140,-26.407,31.327,-36.578
C07898=1013.114,208.575,-138.166,-26.409,31.339,-36.573
C07899=1013.116,208.817,-138.193,-26.410,31.351,-36.567
C07900=1013.117,209.060,-138.220,-26.413,31.363,-36.561
C07901=1013.119,209.301,-138.246,-26.415,31.376,-36.555
C07902=1013.121,209.543,-138.273,-26.416,31.387,-36.549
C07903=1013.122,209.787,-138.300,-26.418,31.400,-36.544
C07904=1013.124,210.028,-138.327,-26.420,31.411,-36.540
C07905=1013.126,210.271,-138.353,-26.422,31.424,-36.532
C07906=1013.128,210.513,-138.380,-26.424,31.436,-36.526
C07907=1013.129,210.756,-138.407,-26.426,31.449,-36.521
C07908=1013.132,210.998,-138.434,-26.428,31.461,-36.515
C07909=1013.132,211.241,-138.460,-26.430,31.472,-36.511
C07910=1013.135,211.484,-138.488,-26.432,31.484,-36.505
C07911=1013.137,211.727,-138.514,-26.434,31.497,-36.499
C07912=1013.138,211.969,-138.541,-26.436,31.508,-36.493
C07913=1013.140,212.213,-138.567,-26.438,31.521,-36.488
C07914=1013.142,212.455,-138.594,-26.440,31.533,-36.482
C07915=1013.144,212.699,-138.622,-26.442,31.544,-36.476
C07916=1013.145,212.943,-138.649,-26.444,31.557,-36.470
C07917=1013.147,213.187,-138.675,-26.446,31.569,-36.465
C07918=1013.149,213.431,-138.702,-26.448,31.580,-36.460
C07919=1013.151,213.675,-138.730,-26.450,31.593,-36.455
C07920=1013.153,213.919,-138.756,-26.452,31.605,-36.449
C07921=1013.155,214.164,-138.783,-26.454,31.617,-36.443
C07922=1013.157,214.408,-138.811,-26.456,31.629,-36.437
C07923=1013.159,214.653,-138.837,-26.457,31.641,-36.432
C07924=1013.160,214.898,-138.865,-26.459,31.654,-36.426
C07925=1013.162,215.143,-138.892,-26.461,31.665,-36.422
C07926=1013.164,215.388,-138.920,-26.463,31.677,-36.416
C07927=1013.166,215.634,-138.947,-26.465,31.688,-36.410
C07928=1013.168,215.878,-138.973,-26.467,31.701,-36.404
C07929=1013.169,216.124,-139.001,-26.469,31.713,-36.399
C07930=1013.172,216.370,-139.028,-26.471,31.726,-36.393
C07931=1013.174,216.618,-139.055,-26.473,31.737,-36.387
C07932=1013.176,216.873,-139.084,-26.475,31.751,-36.380
C07933=1013.178,217.133,-139.113,-26.477,31.763,-36.373
C07934=1013.180,217.397,-139.142,-26.479,31.775,-36.367
C07935=1013.182,217.677,-139.174,-26.481,31.789,-36.361
C07936=1013.185,217.966,-139.205,-26.484,31.804,-36.355
C07937=1013.187,218.260,-139.239,-26.486,31.818,-36.350
C07938=1013.189,218.556,-139.272,-26.488,31.832,-36.345
C07939=1013.192,218.860,-139.305,-26.490,31.847,-36.339
C07940=1013.195,219.155,-139.338,-26.492,31.861,-36.333
C07941=1013.197,219.436,-139.370,-26.495,31.875,-36.326
C07942=1013.199,219.709,-139.400,-26.497,31.888,-36.320
C07943=1013.201,219.969,-139.428,-26.499,31.901,-36.313
C07944=1013.203,220.218,-139.457,-26.501,31.913,-36.307
C07945=1013.205,220.463,-139.484,-26.503,31.924,-36.300
C07946=1013.207,220.709,-139.512,-26.505,31.937,-36.295
C07947=1013.209,220.955,-139.539,-26.506,31.948,-36.289
C07948=1013.211,221.200,-139.566,-26.508,31.960,-36.285
C07949=1013.213,221.446,-139.594,-26.510,31.972,-36.279
C07950=1013.216,221.692,-139.622,-26.512,31.982,-36.274
C07951=1013.218,221.937,-139.649,-26.513,31.992,-36.269
C07952=1013.219,222.183,-139.677,-26.515,32.004,-36.263
C07953=1013.222,222.428,-139.704,-26.517,32.015,-36.258
C07954=1013.223,222.674,-139.732,-26.519,32.027,-36.252
C07955=1013.226,222.920,-139.760,-26.521,32.039,-36.246
C07956=1013.228,223.165,-139.787,-26.523,32.051,-36.241
C07957=1013.230,223.411,-139.814,-26.525,32.063,-36.235
C07958=1013.232,223.657,-139.841,-26.527,32.076,-36.230
C07959=1013.235,223.902,-139.869,-26.529,32.090,-36.223
C07960=1013.237,224.148,-139.897,-26.531,32.102,-36.217
C07961=1013.239,224.394,-139.924,-26.532,32.112,-36.213
C07962=1013.241,224.639,-139.952,-26.534,32.122,-36.207
C07963=1013.243,224.884,-139.980,-26.536,32.133,-36.203
C07964=1013.246,225.131,-140.007,-26.537,32.145,-36.197
C07965=1013.247,225.376,-140.036,-26.539,32.156,-36.193
C07966=1013.250,225.621,-140.063,-26.541,32.168,-36.187
C07967=1013.252,225.867,-140.090,-26.543,32.180,-36.181
C07968=1013.254,226.113,-140.119,-26.545,32.193,-36.176
C07969=1013.256,226.358,-140.146,-26.547,32.206,-36.169
C07970=1013.259,226.604,-140.173,-26.549,32.218,-36.163
C07971=1013.260,226.849,-140.201,-26.551,32.230,-36.157
C07972=1013.263,227.095,-140.229,-26.552,32.241,-36.152
C07973=1013.266,227.340,-140.257,-26.554,32.251,-36.147
C07974=1013.267,227.586,-140.284,-26.556,32.261,-36.143
C07975=1013.270,227.831,-140.312,-26.557,32.273,-36.137
C07976=1013.273,228.077,-140.339,-26.559,32.285,-36.132
C07977=1013.274,228.322,-140.368,-26.561,32.296,-36.126
C07978=1013.277,228.568,-140.395,-26.563,32.309,-36.121
C07979=1013.280,228.813,-140.423,-26.565,32.321,-36.115
C07980=1013.281,229.059,-140.451,-26.567,32.334,-36.108
C07981=1013.284,229.304,-140.479,-26.569,32.347,-36.103
C07982=1013.286,229.550,-140.506,-26.571,32.358,-36.098
C07983=1013.288,229.796,-140.534,-26.572,32.367,-36.093
C07984=1013.290,230.041,-140.562,-26.574,32.378,-36.088
C07985=1013.294,230.287,-140.590,-26.576,32.389,-36.082
C07986=1013.295,230.532,-140.618,-26.577,32.400,-36.077
C07987=1013.297,230.777,-140.645,-26.579,32.412,-36.072
C07988=1013.301,231.023,-140.673,-26.581,32.424,-36.066
C07989=1013.302,231.269,-140.701,-26.583,32.436,-36.060
C07990=1013.305,231.514,-140.729,-26.585,32.449,-36.055
C07991=1013.308,231.759,-140.757,-26.587,32.462,-36.048
C07992=1013.309,232.005,-140.785,-26.589,32.474,-36.042
C07993=1013.312,232.250,-140.812,-26.590,32.483,-36.039
C07994=1013.315,232.496,-140.841,-26.592,32.493,-36.033
C07995=1013.317,232.741,-140.869,-26.593,32.505,-36.027
C07996=1013.319,232.987,-140.896,-26.595,32.516,-36.023
C07997=1013.322,233.232,-140.924,-26.597,32.527,-36.018
C07998=1013.324,233.477,-140.953,-26.599,32.538,-36.012
C07999=1013.326,233.723,-140.980,-26.600,32.551,-36.007
C08000=1013.329,233.968,-141.008,-26.602,32.562,-36.001
C08001=1013.331,234.213,-141.036,-26.604,32.575,-35.995
C08002=1013.334,234.459,-141.065,-26.606,32.589,-35.989
C08003=1013.336,234.705,-141.092,-26.608,32.599,-35.984
C08004=1013.338,234.950,-141.120,-26.609,32.609,-35.979
C08005=1013.341,235.195,-141.148,-26.611,32.619,-35.974
C08006=1013.344,235.441,-141.176,-26.613,32.630,-35.969
C08007=1013.346,235.686,-141.205,-26.614,32.641,-35.963
C08008=1013.349,235.932,-141.233,-26.616,32.652,-35.958
C08009=1013.351,236.177,-141.261,-26.618,32.664,-35.952
C08010=1013.353,236.422,-141.289,-26.620,32.676,-35.946
C08011=1013.356,236.668,-141.317,-26.622,32.688,-35.941
C08012=1013.359,236.913,-141.344,-26.623,32.701,-35.935
C08013=1013.361,237.159,-141.373,-26.625,32.714,-35.929
C08014=1013.363,237.404,-141.401,-26.627,32.724,-35.923
C08015=1013.367,237.649,-141.429,-26.628,32.734,-35.918
C08016=1013.369,237.894,-141.457,-26.630,32.744,-35.914
C08017=1013.371,238.140,-141.486,-26.632,32.754,-35.909
C08018=1013.374,238.385,-141.513,-26.633,32.765,-35.904
C08019=1013.377,238.631,-141.542,-26.635,32.777,-35.898
C08020=1013.379,238.876,-141.570,-26.637,32.788,-35.892
C08021=1013.382,239.121,-141.598,-26.639,32.801,-35.886
C08022=1013.385,239.366,-141.626,-26.640,32.812,-35.880
C08023=1013.387,239.612,-141.655,-26.642,32.825,-35.875
C08024=1013.389,239.857,-141.683,-26.644,32.837,-35.869
C08025=1013.393,240.103,-141.711,-26.646,32.847,-35.864
C08026=1013.395,240.349,-141.739,-26.647,32.857,-35.859
C08027=1013.398,240.593,-141.768,-26.649,32.867,-35.854
C08028=1013.401,240.839,-141.796,-26.650,32.878,-35.849
C08029=1013.403,241.084,-141.825,-26.652,32.889,-35.843
C08030=1013.406,241.329,-141.853,-26.654,32.900,-35.839
C08031=1013.408,241.574,-141.881,-26.656,32.912,-35.833
C08032=1013.411,241.820,-141.909,-26.657,32.923,-35.827
C08033=1013.414,242.066,-141.937,-26.659,32.936,-35.821
C08034=1013.417,242.310,-141.966,-26.661,32.949,-35.815
C08035=1013.420,242.556,-141.994,-26.663,32.960,-35.810
C08036=1013.421,242.801,-142.023,-26.664,32.970,-35.805
C08037=1013.425,243.046,-142.051,-26.666,32.980,-35.800
C08038=1013.428,243.291,-142.080,-26.667,32.990,-35.795
C08039=1013.430,243.537,-142.108,-26.669,33.001,-35.790
C08040=1013.433,243.782,-142.136,-26.671,33.011,-35.783
C08041=1013.435,244.027,-142.164,-26.672,33.022,-35.779
C08042=1013.438,244.272,-142.193,-26.674,33.034,-35.773
C08043=1013.441,244.518,-142.222,-26.676,33.046,-35.767
C08044=1013.444,244.763,-142.249,-26.678,33.059,-35.761
C08045=1013.446,245.008,-142.279,-26.680,33.072,-35.755
C08046=1013.449,245.254,-142.307,-26.681,33.082,-35.750
C08047=1013.452,245.499,-142.335,-26.683,33.092,-35.745
C08048=1013.455,245.744,-142.364,-26.684,33.102,-35.740
C08049=1013.458,245.989,-142.393,-26.686,33.112,-35.735
C08050=1013.461,246.234,-142.421,-26.687,33.121,-35.729
C08051=1013.464,246.479,-142.449,-26.689,33.132,-35.725
C08052=1013.466,246.725,-142.478,-26.690,33.144,-35.719
C08053=1013.470,246.970,-142.507,-26.692,33.155,-35.713
C08054=1013.472,247.215,-142.535,-26.694,33.168,-35.707
C08055=1013.475,247.460,-142.564,-26.696,33.180,-35.702
C08056=1013.478,247.706,-142.592,-26.698,33.193,-35.695
C08057=1013.481,247.950,-142.621,-26.699,33.203,-35.690
C08058=1013.483,248.196,-142.650,-26.701,33.212,-35.686
C08059=1013.486,248.441,-142.678,-26.702,33.222,-35.681
C08060=1013.490,248.687,-142.707,-26.704,33.232,-35.676
C08061=1013.492,248.931,-142.736,-26.705,33.242,-35.669
C08062=1013.495,249.177,-142.764,-26.707,33.253,-35.665
C08063=1013.498,249.422,-142.793,-26.708,33.265,-35.659
C08064=1013.502,249.667,-142.822,-26.710,33.276,-35.653
C08065=1013.503,249.912,-142.850,-26.712,33.289,-35.647
C08066=1013.507,250.157,-142.879,-26.714,33.301,-35.641
C08067=1013.510,250.403,-142.907,-26.716,33.313,-35.636
C08068=1013.513,250.648,-142.937,-26.717,33.322,-35.630
C08069=1013.516,250.893,-142.965,-26.718,33.331,-35.626
C08070=1013.519,251.138,-142.993,-26.720,33.341,-35.621
C08071=1013.521,251.383,-143.023,-26.721,33.351,-35.616
C08072=1013.525,251.628,-143.052,-26.723,33.362,-35.610
C08073=1013.528,251.873,-143.081,-26.724,33.373,-35.605
C08074=1013.530,252.119,-143.109,-26.726,33.384,-35.599
C08075=1013.533,252.363,-143.138,-26.728,33.396,-35.593
C08076=1013.537,252.608,-143.167,-26.730,33.408,-35.588
C08077=1013.539,252.854,-143.195,-26.731,33.421,-35.580
C08078=1013.542,253.099,-143.224,-26.733,33.432,-35.576
C08079=1013.546,253.344,-143.253,-26.734,33.441,-35.570
C08080=1013.549,253.589,-143.283,-26.736,33.450,-35.566
C08081=1013.552,253.834,-143.312,-26.737,33.460,-35.561
C08082=1013.555,254.079,-143.340,-26.739,33.470,-35.556
C08083=1013.557,254.324,-143.369,-26.740,33.480,-35.550
C08084=1013.561,254.569,-143.398,-26.742,33.491,-35.545
C08085=1013.564,254.814,-143.427,-26.744,33.503,-35.539
C08086=1013.567,255.060,-143.456,-26.745,33.514,-35.533
C08087=1013.570,255.305,-143.485,-26.747,33.527,-35.528
C08088=1013.574,255.550,-143.514,-26.749,33.539,-35.521
C08089=1013.576,255.795,-143.543,-26.750,33.549,-35.515
C08090=1013.580,256.040,-143.572,-26.752,33.558,-35.512
C08091=1013.583,256.285,-143.601,-26.753,33.567,-35.506
C08092=1013.586,256.530,-143.631,-26.754,33.577,-35.501
C08093=1013.589,256.775,-143.659,-26.756,33.587,-35.496
C08094=1013.593,257.020,-143.688,-26.757,33.597,-35.491
C08095=1013.595,257.265,-143.718,-26.759,33.609,-35.485
C08096=1013.599,257.510,-143.747,-26.761,33.621,-35.479
C08097=1013.602,257.755,-143.775,-26.762,33.632,-35.473
C08098=1013.604,258.000,-143.805,-26.764,33.645,-35.468
C08099=1013.608,258.245,-143.834,-26.766,33.658,-35.461
C08100=1013.621,259.470,-143.986,-26.819,33.830,-34.398
C08101=1013.623,259.875,-144.040,-26.834,33.872,-34.047
C08102=1013.623,260.267,-144.091,-26.853,33.951,-33.694
C08103=1013.623,260.659,-144.145,-26.869,34.014,-33.345
C08104=1013.623,261.051,-144.201,-26.884,34.066,-32.999
C08105=1013.621,261.468,-144.261,-26.904,34.165,-32.615
C08106=1013.621,261.495,-144.265,-26.905,34.173,-32.590
C08107=1013.619,261.899,-144.325,-26.920,34.232,-32.229
C08108=1013.615,262.304,-144.386,-26.937,34.313,-31.862
C08109=1013.611,262.708,-144.449,-26.950,34.363,-31.502
C08110=1013.605,263.112,-144.513,-26.966,34.455,-31.130
C08111=1013.599,263.516,-144.579,-26.979,34.511,-30.766
C08112=1013.592,263.920,-144.646,-26.992,34.584,-30.397
C08113=1013.583,264.324,-144.713,-27.008,34.691,-30.017
C08114=1013.574,264.728,-144.784,-27.018,34.737,-29.656
C08115=1013.564,265.132,-144.854,-27.031,34.828,-29.278
C08116=1013.552,265.536,-144.927,-27.044,34.924,-28.900
C08117=1013.541,265.939,-145.000,-27.055,35.006,-28.525
C08118=1013.528,266.343,-145.076,-27.065,35.079,-28.151
C08119=1013.514,266.745,-145.153,-27.075,35.162,-27.773
C08120=1013.499,267.149,-145.231,-27.085,35.263,-27.389
C08121=1013.484,267.552,-145.311,-27.093,35.326,-27.015
C08122=1013.466,267.954,-145.392,-27.102,35.432,-26.627
C08123=1013.449,268.357,-145.475,-27.109,35.519,-26.243
C08124=1013.430,268.759,-145.559,-27.115,35.600,-25.860
C08125=1013.409,269.161,-145.643,-27.122,35.725,-25.463
C08126=1013.388,269.563,-145.730,-27.127,35.811,-25.075
C08127=1013.367,269.965,-145.818,-27.132,35.920,-24.681
C08128=1013.345,270.367,-145.908,-27.136,35.994,-24.294
C08129=1013.320,270.768,-145.998,-27.139,36.112,-23.895
C08130=1013.296,271.169,-146.091,-27.141,36.202,-23.501
C08131=1013.270,271.571,-146.186,-27.142,36.308,-23.102
C08132=1013.243,271.972,-146.281,-27.142,36.422,-22.700
C08133=1013.215,272.372,-146.378,-27.142,36.517,-22.302
C08134=1013.186,272.772,-146.475,-27.140,36.653,-21.889
C08135=1013.156,273.173,-146.575,-27.138,36.755,-21.484
C08136=1013.125,273.574,-146.677,-27.134,36.862,-21.077
C08137=1013.093,273.973,-146.780,-27.129,36.975,-20.665
C08138=1013.061,274.373,-146.883,-27.123,37.106,-20.245
C08139=1013.026,274.772,-146.989,-27.116,37.225,-19.825
C08140=1012.992,275.171,-147.097,-27.108,37.339,-19.406
C08141=1012.956,275.570,-147.205,-27.098,37.466,-18.981
C08142=1012.918,275.969,-147.315,-27.087,37.595,-18.552
C08143=1012.880,276.368,-147.427,-27.075,37.727,-18.120
C08144=1012.841,276.766,-147.540,-27.062,37.854,-17.687
C08145=1012.800,277.164,-147.655,-27.046,37.998,-17.247
C08146=1012.759,277.561,-147.772,-27.031,38.109,-16.814
C08147=1012.716,277.958,-147.889,-27.011,38.268,-16.364
C08148=1012.673,278.356,-148.009,-26.991,38.409,-15.917
C08149=1012.629,278.752,-148.131,-26.971,38.537,-15.471
C08150=1012.582,279.148,-148.253,-26.946,38.689,-15.016
C08151=1012.536,279.545,-148.377,-26.922,38.832,-14.559
C08152=1012.487,279.940,-148.503,-26.894,38.990,-14.092
C08153=1012.439,280.335,-148.630,-26.863,39.152,-13.621
C08154=1012.388,280.730,-148.759,-26.831,39.313,-13.145
C08155=1012.337,281.124,-148.889,-26.798,39.468,-12.665
C08156=1012.284,281.518,-149.021,-26.759,39.647,-12.176
C08157=1012.230,281.912,-149.155,-26.720,39.816,-11.682
C08158=1012.175,282.306,-149.290,-26.678,39.991,-11.184
C08159=1012.119,282.698,-149.427,-26.633,40.164,-10.680
C08160=1012.062,283.091,-149.567,-26.586,40.342,-10.169
C08161=1012.003,283.482,-149.706,-26.533,40.540,-9.648
C08162=1011.944,283.874,-149.848,-26.478,40.729,-9.124
C08163=1011.883,284.265,-149.992,-26.421,40.916,-8.596
C08164=1011.821,284.655,-150.138,-26.362,41.102,-8.062
C08165=1011.757,285.045,-150.285,-26.294,41.317,-7.515
C08166=1011.692,285.435,-150.434,-26.225,41.525,-6.963
C08167=1011.627,285.823,-150.585,-26.152,41.732,-6.403
C08168=1011.560,286.212,-150.738,-26.076,41.936,-5.835
C08169=1011.491,286.599,-150.890,-25.990,42.171,-5.252
C08170=1011.422,286.986,-151.047,-25.906,42.382,-4.665
C08171=1011.387,287.180,-151.126,-25.858,42.503,-4.364
C08172=1011.350,287.373,-151.205,-25.807,42.634,-4.060
C08173=1011.314,287.565,-151.284,-25.760,42.745,-3.758
C08174=1011.278,287.759,-151.365,-25.708,42.870,-3.450
C08175=1011.241,287.951,-151.446,-25.659,42.982,-3.144
C08176=1011.205,288.144,-151.527,-25.607,43.098,-2.834
C08177=1011.167,288.336,-151.608,-25.550,43.230,-2.517
C08178=1011.129,288.528,-151.690,-25.492,43.360,-2.199
C08179=1011.091,288.720,-151.772,-25.433,43.487,-1.879
C08180=1011.053,288.912,-151.855,-25.375,43.611,-1.558
C08181=1011.013,289.103,-151.938,-25.312,43.742,-1.232
C08182=1010.975,289.295,-152.022,-25.250,43.869,-0.904
C08183=1010.936,289.486,-152.107,-25.185,44.000,-0.573
C08184=1010.896,289.677,-152.191,-25.117,44.136,-0.237
C08185=1010.855,289.868,-152.277,-25.050,44.264,0.100
C08186=1010.815,290.059,-152.362,-24.977,44.406,0.444
C08187=1010.774,290.248,-152.448,-24.905,44.542,0.788
C08188=1010.733,290.439,-152.536,-24.831,44.677,1.136
C08189=1010.691,290.629,-152.622,-24.750,44.829,1.491
C08190=1010.649,290.819,-152.710,-24.671,44.968,1.846
C08191=1010.607,291.008,-152.798,-24.587,45.118,2.207
C08192=1010.565,291.198,-152.888,-24.506,45.255,2.568
C08193=1010.522,291.387,-152.977,-24.417,45.407,2.935
C08194=1010.479,291.576,-153.068,-24.330,45.548,3.304
C08195=1010.435,291.765,-153.158,-24.241,45.692,3.677
C08196=1010.390,291.954,-153.248,-24.142,45.855,4.058
C08197=1010.345,292.141,-153.340,-24.043,46.013,4.442
C08198=1010.301,292.329,-153.432,-23.942,46.171,4.829
C08199=1010.256,292.518,-153.524,-23.840,46.324,5.219
C08200=1010.210,292.705,-153.617,-23.733,46.485,5.616
C08201=1010.164,292.893,-153.711,-23.625,46.643,6.015
C08202=1010.118,293.079,-153.805,-23.513,46.805,6.419
C08203=1010.070,293.266,-153.899,-23.394,46.975,6.831
C08204=1010.024,293.453,-153.994,-23.278,47.134,7.243
C08205=1009.976,293.639,-154.090,-23.151,47.310,7.666
C08206=1009.928,293.826,-154.186,-23.028,47.472,8.087
C08207=1009.879,294.011,-154.283,-22.897,47.647,8.516
C08208=1009.830,294.197,-154.380,-22.762,47.822,8.950
C08209=1009.781,294.382,-154.478,-22.622,48.001,9.391
C08210=1009.732,294.566,-154.576,-22.485,48.168,9.831
C08211=1009.681,294.752,-154.676,-22.336,48.353,10.283
C08212=1009.631,294.936,-154.775,-22.191,48.522,10.734
C08213=1009.580,295.120,-154.876,-22.037,48.704,11.195
C08214=1009.528,295.305,-154.976,-21.871,48.900,11.664
C08215=1009.477,295.488,-155.077,-21.710,49.081,12.135
C08216=1009.425,295.671,-155.180,-21.542,49.268,12.613
C08217=1009.372,295.854,-155.282,-21.368,49.457,13.097
C08218=1009.319,296.037,-155.385,-21.192,49.644,13.585
///RCONF 0,0,0,0,0,0,0,0,0,0,0,0,0,0,0,0,0,0,0,0,0,0,0,0
C08219=1009.266,296.219,-155.489,-21.008,49.838,14.081
C08220=1009.213,296.402,-155.593,-20.821,50.028,14.582
C08221=1009.158,296.583,-155.698,-20.628,50.221,15.091
C08222=1009.104,296.764,-155.803,-20.424,50.425,15.608
C08223=1009.049,296.946,-155.909,-20.226,50.611,16.126
C08224=1008.992,297.126,-156.016,-20.012,50.816,16.657
C08225=1008.937,297.307,-156.123,-19.794,51.019,17.192
C08226=1008.880,297.488,-156.231,-19.575,51.214,17.733
C08227=1008.823,297.667,-156.340,-19.338,51.428,18.287
C08228=1008.765,297.848,-156.449,-19.102,51.633,18.845
C08229=1008.708,298.027,-156.558,-18.856,51.845,19.411
C08230=1008.650,298.205,-156.668,-18.612,52.043,19.979
C08231=1008.591,298.383,-156.780,-18.352,52.256,20.562
C08232=1008.531,298.562,-156.891,-18.083,52.472,21.153
C08233=1008.471,298.740,-157.003,-17.809,52.687,21.752
C08234=1008.412,298.917,-157.115,-17.532,52.895,22.355
C08235=1008.350,299.094,-157.230,-17.244,53.109,22.968
C08236=1008.290,299.271,-157.343,-16.948,53.324,23.590
C08237=1008.228,299.448,-157.458,-16.646,53.537,24.220
C08238=1008.166,299.623,-157.573,-16.332,53.755,24.861
C08239=1008.103,299.799,-157.690,-16.011,53.971,25.511
C08240=1008.040,299.974,-157.806,-15.683,54.186,26.168
C08241=1007.977,300.148,-157.924,-15.334,54.414,26.841
C08242=1007.914,300.323,-158.042,-14.991,54.626,27.516
C08243=1007.848,300.497,-158.161,-14.624,54.854,28.209
C08244=1007.784,300.671,-158.279,-14.262,55.066,28.903
C08245=1007.718,300.844,-158.399,-13.874,55.295,29.618
C08246=1007.652,301.016,-158.520,-13.487,55.512,30.335
C08247=1007.586,301.189,-158.641,-13.089,55.730,31.065
C08248=1007.518,301.360,-158.763,-12.673,55.954,31.809
C08249=1007.451,301.532,-158.886,-12.259,56.165,32.558
C08250=1007.383,301.703,-159.009,-11.822,56.387,33.325
C08251=1007.315,301.873,-159.133,-11.370,56.612,34.103
C08252=1007.246,302.043,-159.257,-10.909,56.834,34.893
C08253=1007.177,302.214,-159.384,-10.444,57.047,35.689
C08254=1007.106,302.383,-159.509,-9.963,57.264,36.498
C08255=1007.037,302.552,-159.635,-9.470,57.478,37.320
C08256=1006.966,302.720,-159.763,-8.966,57.690,38.154
C08257=1006.894,302.887,-159.890,-8.446,57.903,39.002
C08258=1006.822,303.055,-160.020,-7.913,58.114,39.864
C08259=1006.750,303.221,-160.149,-7.371,58.320,40.735
C08260=1006.676,303.388,-160.278,-6.799,58.537,41.628
C08261=1006.604,303.555,-160.409,-6.235,58.735,42.521
C08262=1006.529,303.720,-160.540,-5.636,58.946,43.442
C08263=1006.455,303.884,-160.673,-5.045,59.140,44.363
C08264=1006.380,304.049,-160.805,-4.417,59.345,45.310
C08265=1006.304,304.212,-160.939,-3.788,59.539,46.265
C08266=1006.228,304.376,-161.073,-3.145,59.728,47.232
C08267=1006.151,304.539,-161.207,-2.482,59.919,48.216
C08268=1006.074,304.701,-161.343,-1.819,60.098,49.205
C08269=1005.997,304.863,-161.479,-1.131,60.279,50.212
C08270=1005.918,305.023,-161.616,-0.416,60.463,51.239
C08271=1005.839,305.184,-161.753,0.303,60.637,52.274
C08272=1005.760,305.344,-161.891,1.028,60.802,53.319
C08273=1005.681,305.504,-162.031,1.776,60.967,54.381
C08274=1005.601,305.662,-162.169,2.534,61.125,55.453
C08275=1005.520,305.821,-162.310,3.309,61.278,56.542
C08276=1005.439,305.979,-162.451,4.097,61.427,57.641
C08277=1005.357,306.135,-162.593,4.899,61.569,58.754
C08278=1005.275,306.292,-162.735,5.713,61.705,59.880
C08279=1005.192,306.448,-162.877,6.561,61.844,61.027
C08280=1005.109,306.603,-163.020,7.390,61.962,62.171
C08281=1005.025,306.758,-163.165,8.260,62.085,63.340
C08282=1004.940,306.912,-163.309,9.126,62.195,64.514
C08283=1004.856,307.066,-163.455,10.011,62.301,65.700
C08284=1004.770,307.219,-163.601,10.917,62.404,66.900
C08285=1004.684,307.371,-163.748,11.823,62.496,68.103
C08286=1004.597,307.523,-163.896,12.730,62.575,69.311
C08287=1004.511,307.674,-164.044,13.658,62.653,70.529
C08288=1004.424,307.824,-164.193,14.581,62.717,71.749
C08289=1004.336,307.973,-164.342,15.516,62.776,72.977
C08290=1004.247,308.123,-164.492,16.490,62.836,74.228
C08291=1004.165,308.259,-164.632,17.370,62.876,75.375
C08292=1004.082,308.396,-164.771,18.264,62.912,76.528
C08293=1004.000,308.532,-164.912,19.155,62.936,77.684
C08294=1003.916,308.668,-165.052,20.063,62.958,78.847
C08295=1004.326,308.744,-165.526,5.994,57.263,73.789
C08296=1004.428,308.576,-165.350,4.899,57.107,72.274
C08297=1004.532,308.409,-165.177,3.803,56.929,70.768
C08298=1004.634,308.240,-165.004,2.734,56.742,69.279
C08299=1004.735,308.071,-164.832,1.687,56.543,67.809
C08300=1004.825,307.922,-164.683,0.767,56.348,66.529
C08301=1004.912,307.772,-164.533,-0.116,56.156,65.268
C08302=1004.999,307.622,-164.384,-0.976,55.958,64.026
C08303=1005.086,307.471,-164.236,-1.838,55.743,62.786
C08304=1005.172,307.319,-164.088,-2.667,55.527,61.571
C08305=1005.258,307.167,-163.941,-3.491,55.298,60.364
C08306=1005.344,307.014,-163.795,-4.306,55.057,59.166
C08307=1005.429,306.861,-163.650,-5.095,54.813,57.987
C08308=1005.513,306.706,-163.505,-5.862,54.566,56.824
C08309=1005.597,306.552,-163.361,-6.624,54.303,55.672
C08310=1005.679,306.397,-163.217,-7.345,54.050,54.548
C08311=1005.763,306.241,-163.075,-8.077,53.772,53.425
C08312=1005.845,306.084,-162.933,-8.770,53.502,52.330
C08313=1005.927,305.926,-162.791,-9.451,53.223,51.248
C08314=1006.008,305.769,-162.650,-10.114,52.940,50.182
C08315=1006.088,305.611,-162.510,-10.758,52.654,49.132
C08316=1006.168,305.452,-162.371,-11.385,52.363,48.098
C08317=1006.248,305.293,-162.232,-11.999,52.066,47.078
C08318=1006.327,305.132,-162.094,-12.588,51.771,46.077
C08319=1006.406,304.972,-161.957,-13.169,51.466,45.085
C08320=1006.484,304.811,-161.820,-13.741,51.153,44.107
C08321=1006.562,304.649,-161.685,-14.287,50.844,43.148
C08322=1006.639,304.486,-161.548,-14.810,50.541,42.204
C08323=1006.715,304.324,-161.414,-15.328,50.224,41.271
C08324=1006.792,304.160,-161.279,-15.826,49.912,40.354
C08325=1006.867,303.997,-161.147,-16.310,49.597,39.449
C08326=1006.942,303.832,-161.013,-16.790,49.269,38.552
C08327=1007.016,303.668,-160.882,-17.238,48.959,37.678
C08328=1007.090,303.502,-160.751,-17.689,48.629,36.809
C08329=1007.164,303.336,-160.620,-18.109,48.316,35.963
C08330=1007.238,303.170,-160.490,-18.533,47.985,35.121
C08331=1007.310,303.003,-160.361,-18.931,47.667,34.296
C08332=1007.382,302.836,-160.233,-19.318,47.346,33.485
C08333=1007.453,302.668,-160.104,-19.694,47.024,32.684
C08334=1007.524,302.500,-159.977,-20.055,46.705,31.896
C08335=1007.594,302.331,-159.851,-20.406,46.386,31.120
C08336=1007.664,302.162,-159.724,-20.746,46.065,30.353
C08337=1007.733,301.992,-159.600,-21.071,45.750,29.599
C08338=1007.802,301.821,-159.475,-21.391,45.428,28.853
C08339=1007.871,301.652,-159.351,-21.704,45.103,28.116
C08340=1007.938,301.480,-159.228,-22.002,44.783,27.390
C08341=1008.005,301.308,-159.105,-22.281,44.479,26.681
C08342=1008.073,301.137,-158.984,-22.561,44.159,25.973
C08343=1008.139,300.964,-158.862,-22.825,43.851,25.281
C08344=1008.204,300.792,-158.741,-23.080,43.544,24.597
C08345=1008.271,300.619,-158.623,-23.335,43.225,23.918
C08346=1008.335,300.445,-158.502,-23.568,42.928,23.257
C08347=1008.400,300.272,-158.384,-23.803,42.614,22.596
C08348=1008.463,300.097,-158.266,-24.021,42.318,21.951
C08349=1008.527,299.922,-158.149,-24.241,42.008,21.307
C08350=1008.590,299.747,-158.032,-24.445,41.713,20.679
C08351=1008.652,299.571,-157.917,-24.642,41.419,20.056
C08352=1008.714,299.395,-157.801,-24.833,41.125,19.442
C08353=1008.776,299.219,-157.686,-25.015,40.837,18.837
///RCONF 0,0,0,0,1,0,0,0,0,0,0,0,0,0,0,0,0,0,0,0,0,0,0,0
C08354=1008.837,299.042,-157.572,-25.191,40.548,18.237
C08355=1008.898,298.865,-157.459,-25.361,40.262,17.646
C08356=1008.958,298.688,-157.346,-25.521,39.984,17.065
C08357=1009.017,298.510,-157.234,-25.680,39.700,16.487
C08358=1009.076,298.332,-157.123,-25.834,39.415,15.914
C08359=1009.136,298.153,-157.012,-25.980,39.136,15.350
C08360=1009.194,297.975,-156.901,-26.113,38.875,14.798
C08361=1009.252,297.795,-156.792,-26.248,38.599,14.248
C08362=1009.309,297.615,-156.682,-26.376,38.332,13.705
C08363=1009.366,297.436,-156.574,-26.503,38.057,13.167
C08364=1009.423,297.255,-156.467,-26.616,37.804,12.639
C08365=1009.478,297.075,-156.359,-26.729,37.543,12.114
C08366=1009.534,296.894,-156.253,-26.839,37.281,11.594
C08367=1009.589,296.713,-156.146,-26.936,37.042,11.089
C08368=1009.644,296.531,-156.041,-27.036,36.785,10.581
C08369=1009.698,296.350,-155.937,-27.129,36.540,10.081
C08370=1009.752,296.167,-155.832,-27.217,36.298,9.588
C08371=1009.805,295.985,-155.729,-27.303,36.055,9.099
C08372=1009.858,295.802,-155.626,-27.383,35.820,8.617
C08373=1009.911,295.619,-155.523,-27.461,35.584,8.139
C08374=1009.962,295.436,-155.422,-27.534,35.352,7.666
C08375=1010.014,295.252,-155.320,-27.602,35.127,7.201
C08376=1010.066,295.068,-155.219,-27.674,34.884,6.733
C08377=1010.117,294.884,-155.120,-27.737,34.661,6.276
C08378=1010.167,294.700,-155.019,-27.793,34.453,5.828
C08379=1010.217,294.515,-154.921,-27.851,34.228,5.379
C08380=1010.266,294.330,-154.823,-27.902,34.022,4.940
C08381=1010.316,294.145,-154.724,-27.954,33.804,4.500
C08382=1010.364,293.959,-154.627,-28.003,33.591,4.064
C08383=1010.413,293.773,-154.531,-28.049,33.380,3.635
C08384=1010.460,293.588,-154.435,-28.089,33.184,3.213
C08385=1010.508,293.401,-154.340,-28.131,32.973,2.790
C08386=1010.556,293.214,-154.244,-28.166,32.783,2.376
C08387=1010.603,293.028,-154.149,-28.202,32.579,1.962
C08388=1010.649,292.840,-154.056,-28.234,32.387,1.554
C08389=1010.695,292.653,-153.961,-28.264,32.199,1.152
C08390=1010.740,292.465,-153.869,-28.292,32.009,0.753
C08391=1010.785,292.278,-153.777,-28.317,31.827,0.359
C08392=1010.830,292.089,-153.684,-28.341,31.642,-0.033
C08393=1010.875,291.902,-153.594,-28.364,31.455,-0.424
C08394=1010.920,291.713,-153.503,-28.386,31.266,-0.810
C08395=1010.962,291.524,-153.412,-28.403,31.099,-1.187
C08396=1011.006,291.335,-153.323,-28.417,30.935,-1.561
C08397=1011.049,291.146,-153.233,-28.433,30.758,-1.936
C08398=1011.091,290.956,-153.144,-28.444,30.599,-2.302
C08399=1011.134,290.767,-153.056,-28.456,30.428,-2.670
C08400=1011.176,290.577,-152.968,-28.465,30.268,-3.031
C08401=1011.217,290.387,-152.881,-28.475,30.094,-3.396
C08402=1011.258,290.197,-152.795,-28.481,29.939,-3.750
C08403=1011.300,290.007,-152.708,-28.486,29.784,-4.103
C08404=1011.340,289.816,-152.623,-28.491,29.623,-4.455
C08405=1011.380,289.625,-152.537,-28.493,29.479,-4.798
C08406=1011.420,289.433,-152.452,-28.495,29.324,-5.144
C08407=1011.459,289.243,-152.368,-28.495,29.177,-5.483
C08408=1011.498,289.051,-152.284,-28.493,29.035,-5.820
C08409=1011.537,288.860,-152.201,-28.492,28.887,-6.156
C08410=1011.575,288.668,-152.119,-28.488,28.750,-6.486
C08411=1011.613,288.476,-152.036,-28.484,28.608,-6.814
C08412=1011.651,288.284,-151.955,-28.479,28.464,-7.143
C08413=1011.689,288.092,-151.873,-28.474,28.318,-7.470
C08414=1011.726,287.899,-151.791,-28.466,28.190,-7.790
C08415=1011.761,287.707,-151.711,-28.457,28.068,-8.104
C08416=1011.798,287.514,-151.630,-28.449,27.930,-8.424
C08417=1011.833,287.321,-151.551,-28.438,27.811,-8.734
C08418=1011.905,286.934,-151.394,-28.418,27.534,-9.364
C08419=1011.975,286.547,-151.238,-28.390,27.307,-9.969
C08420=1012.044,286.160,-151.084,-28.363,27.054,-10.577
C08421=1012.111,285.772,-150.931,-28.331,26.837,-11.165
C08422=1012.176,285.383,-150.780,-28.297,26.617,-11.746
C08423=1012.241,284.993,-150.632,-28.261,26.397,-12.321
C08424=1012.305,284.604,-150.484,-28.224,26.170,-12.894
C08425=1012.366,284.213,-150.339,-28.183,25.978,-13.449
C08426=1012.427,283.822,-150.195,-28.141,25.784,-14.001
C08427=1012.486,283.431,-150.053,-28.096,25.589,-14.548
C08428=1012.545,283.039,-149.913,-28.051,25.385,-15.094
C08429=1012.602,282.646,-149.775,-28.003,25.205,-15.628
C08430=1012.658,282.254,-149.637,-27.954,25.030,-16.155
C08431=1012.713,281.861,-149.502,-27.904,24.854,-16.680
C08432=1012.767,281.467,-149.368,-27.852,24.684,-17.197
C08433=1012.820,281.073,-149.236,-27.799,24.506,-17.713
C08434=1012.871,280.678,-149.106,-27.745,24.357,-18.215
C08435=1012.921,280.284,-148.977,-27.690,24.197,-18.716
C08436=1012.971,279.888,-148.851,-27.634,24.040,-19.214
C08437=1013.019,279.493,-148.725,-27.577,23.887,-19.705
C08438=1013.065,279.097,-148.601,-27.520,23.752,-20.185
C08439=1013.111,278.701,-148.478,-27.462,23.605,-20.666
C08440=1013.155,278.304,-148.357,-27.403,23.486,-21.135
C08441=1013.199,277.907,-148.238,-27.343,23.354,-21.606
C08442=1013.242,277.510,-148.121,-27.282,23.205,-22.083
C08443=1013.283,277.112,-148.003,-27.222,23.105,-22.537
C08444=1013.324,276.715,-147.889,-27.159,22.972,-23.004
C08445=1013.363,276.316,-147.776,-27.097,22.857,-23.460
C08446=1013.401,275.918,-147.665,-27.033,22.739,-23.918
C08447=1013.438,275.520,-147.554,-26.969,22.622,-24.371
C08448=1013.474,275.121,-147.445,-26.905,22.510,-24.822
C08449=1013.509,274.721,-147.338,-26.841,22.411,-25.264
C08450=1013.543,274.322,-147.232,-26.776,22.307,-25.707
C08451=1013.577,273.922,-147.128,-26.709,22.192,-26.154
C08452=1013.609,273.523,-147.026,-26.644,22.096,-26.590
C08453=1013.639,273.122,-146.924,-26.579,22.005,-27.022
C08454=1013.668,272.722,-146.823,-26.514,21.923,-27.448
C08455=1013.749,271.566,-146.544,-26.318,21.640,-28.693
C08456=1013.774,271.188,-146.457,-26.259,21.599,-29.073
C08457=1013.797,270.810,-146.368,-26.201,21.560,-29.450
C08458=1013.814,270.531,-146.305,-26.158,21.533,-29.728
C08459=1013.830,270.254,-146.242,-26.115,21.507,-30.003
C08460=1013.845,269.975,-146.180,-26.072,21.483,-30.277
C08461=1013.861,269.698,-146.118,-26.030,21.459,-30.551
C08462=1013.874,269.453,-146.066,-25.992,21.439,-30.789
C08463=1013.887,269.209,-146.013,-25.955,21.420,-31.029
C08464=1013.900,268.965,-145.961,-25.918,21.402,-31.266
C08465=1013.911,268.720,-145.909,-25.881,21.386,-31.502
C08466=1013.925,268.442,-145.851,-25.839,21.367,-31.772
C08467=1013.937,268.164,-145.793,-25.797,21.350,-32.039
C08468=1013.949,267.885,-145.736,-25.755,21.334,-32.305
C08469=1013.962,267.607,-145.681,-25.714,21.319,-32.571
C08470=1013.972,267.361,-145.632,-25.677,21.306,-32.805
C08471=1013.980,267.116,-145.583,-25.641,21.295,-33.037
C08472=1013.990,266.871,-145.535,-25.604,21.284,-33.268
C08473=1013.999,266.626,-145.488,-25.568,21.275,-33.499
C08474=1014.009,266.347,-145.435,-25.527,21.264,-33.760
C08475=1014.017,266.069,-145.383,-25.487,21.254,-34.021
C08476=1014.027,265.789,-145.331,-25.446,21.246,-34.279
C08477=1014.034,265.510,-145.280,-25.406,21.239,-34.538
C08478=1014.041,265.265,-145.235,-25.370,21.233,-34.766
C08479=1014.048,265.018,-145.192,-25.335,21.229,-34.991
C08480=1014.055,264.772,-145.148,-25.300,21.225,-35.219
C08481=1014.061,264.526,-145.106,-25.265,21.221,-35.444
C08482=1014.066,264.247,-145.056,-25.226,21.219,-35.699
C08483=1014.073,263.969,-145.010,-25.186,21.217,-35.952
C08484=1014.079,263.690,-144.964,-25.147,21.216,-36.205
C08485=1014.083,263.411,-144.917,-25.108,21.215,-36.458
C08486=1014.086,263.164,-144.877,-25.074,21.216,-36.681
C08487=1014.090,262.917,-144.838,-25.040,21.218,-36.903
C08488=1014.093,262.670,-144.798,-25.006,21.220,-37.124
C08489=1014.096,262.423,-144.760,-24.973,21.223,-37.345
C08490=1014.098,262.144,-144.717,-24.935,21.227,-37.593
C08491=1014.101,261.865,-144.675,-24.897,21.232,-37.841
C08492=1014.103,261.586,-144.634,-24.860,21.238,-38.088
C08493=1014.104,261.307,-144.592,-24.823,21.244,-38.335
C08494=1014.106,261.059,-144.557,-24.790,21.252,-38.553
C08495=1014.106,260.812,-144.522,-24.758,21.259,-38.770
C08496=1014.107,260.564,-144.487,-24.726,21.267,-38.987
C08497=1014.105,260.316,-144.452,-24.693,21.275,-39.204
C08498=1014.106,260.036,-144.415,-24.658,21.287,-39.446
C08499=1014.105,259.757,-144.377,-24.622,21.298,-39.688
C08500=1014.104,259.477,-144.341,-24.587,21.310,-39.930
C08501=1014.101,259.198,-144.304,-24.552,21.323,-40.170
C08502=1014.090,258.206,-144.182,-24.430,21.374,-41.010
C08503=1014.086,257.858,-144.140,-24.430,21.376,-41.012
C08504=1014.082,257.512,-144.099,-24.430,21.375,-41.016
C08505=1014.078,257.165,-144.058,-24.429,21.376,-41.019
C08506=1014.073,256.817,-144.017,-24.429,21.376,-41.023
C08507=1014.070,256.570,-143.987,-24.428,21.376,-41.027
C08508=1014.067,256.322,-143.958,-24.428,21.376,-41.028
C08509=1014.063,256.073,-143.929,-24.428,21.377,-41.031
C08510=1014.060,255.825,-143.899,-24.427,21.376,-41.034
C08511=1014.055,255.437,-143.853,-24.427,21.377,-41.038
C08512=1014.051,255.049,-143.806,-24.426,21.377,-41.042
C08513=1014.046,254.661,-143.761,-24.426,21.378,-41.045
C08514=1014.041,254.273,-143.715,-24.425,21.377,-41.049
C08515=1014.039,254.024,-143.686,-24.424,21.378,-41.052
C08516=1014.034,253.776,-143.656,-24.424,21.378,-41.054
C08517=1014.032,253.528,-143.627,-24.424,21.378,-41.058
C08518=1014.029,253.280,-143.598,-24.423,21.378,-41.060
C08519=1014.025,253.031,-143.568,-24.423,21.378,-41.061
C08520=1014.023,252.783,-143.539,-24.423,21.378,-41.065
C08521=1014.020,252.535,-143.510,-24.422,21.379,-41.067
C08522=1014.017,252.287,-143.480,-24.422,21.379,-41.069
C08523=1014.014,252.039,-143.452,-24.421,21.378,-41.072
C08524=1014.011,251.790,-143.422,-24.421,21.379,-41.074
C08525=1014.008,251.541,-143.393,-24.421,21.380,-41.076
C08526=1014.005,251.294,-143.363,-24.421,21.380,-41.078
C08527=1014.002,251.050,-143.335,-24.420,21.380,-41.082
C08528=1013.999,250.807,-143.306,-24.420,21.380,-41.084
C08529=1013.996,250.564,-143.277,-24.420,21.380,-41.085
C08530=1013.993,250.321,-143.248,-24.419,21.380,-41.089
C08531=1013.990,250.077,-143.221,-24.419,21.380,-41.091
C08532=1013.987,249.834,-143.192,-24.419,21.381,-41.093
C08533=1013.985,249.592,-143.163,-24.418,21.381,-41.095
C08534=1013.981,249.348,-143.135,-24.418,21.381,-41.098
C08535=1013.979,249.099,-143.106,-24.418,21.381,-41.100
C08536=1013.975,248.851,-143.077,-24.417,21.381,-41.102
C08537=1013.973,248.603,-143.047,-24.417,21.381,-41.104
C08538=1013.970,248.355,-143.018,-24.417,21.381,-41.107
C08539=1013.967,248.107,-142.989,-24.416,21.381,-41.109
C08540=1013.965,247.859,-142.960,-24.416,21.382,-41.111
C08541=1013.961,247.610,-142.931,-24.416,21.382,-41.113
C08542=1013.958,247.362,-142.901,-24.415,21.382,-41.117
C08543=1013.955,247.113,-142.873,-24.415,21.382,-41.118
C08544=1013.953,246.865,-142.844,-24.415,21.382,-41.120
C08545=1013.949,246.617,-142.815,-24.414,21.383,-41.122
C08546=1013.947,246.368,-142.786,-24.414,21.382,-41.126
C08547=1013.944,246.120,-142.756,-24.414,21.382,-41.127
C08548=1013.941,245.872,-142.728,-24.413,21.383,-41.129
C08549=1013.939,245.623,-142.699,-24.413,21.384,-41.132
C08550=1013.936,245.375,-142.670,-24.413,21.384,-41.134
C08551=1013.933,245.127,-142.641,-24.412,21.384,-41.137
C08552=1013.930,244.878,-142.613,-24.412,21.384,-41.139
C08553=1013.928,244.630,-142.583,-24.412,21.384,-41.141
C08554=1013.924,244.382,-142.555,-24.412,21.384,-41.143
C08555=1013.922,244.139,-142.526,-24.411,21.384,-41.144
C08556=1013.919,243.896,-142.498,-24.411,21.384,-41.148
C08557=1013.917,243.652,-142.470,-24.411,21.384,-41.150
C08558=1013.914,243.410,-142.441,-24.410,21.384,-41.151
C08559=1013.911,243.166,-142.414,-24.410,21.385,-41.153
C08560=1013.909,242.923,-142.385,-24.410,21.385,-41.155
C08561=1013.906,242.680,-142.357,-24.410,21.385,-41.157
C08562=1013.903,242.437,-142.328,-24.409,21.385,-41.159
C08563=1013.900,242.189,-142.300,-24.409,21.385,-41.162
C08564=1013.898,241.941,-142.271,-24.408,21.385,-41.164
C08565=1013.895,241.693,-142.243,-24.408,21.385,-41.166
C08566=1013.893,241.444,-142.214,-24.408,21.386,-41.168
C08567=1013.890,241.196,-142.186,-24.408,21.386,-41.170
C08568=1013.887,240.947,-142.156,-24.407,21.386,-41.172
C08569=1013.884,240.699,-142.128,-24.407,21.386,-41.174
C08570=1013.882,240.450,-142.099,-24.407,21.386,-41.177
C08571=1013.879,240.203,-142.070,-24.406,21.386,-41.179
C08572=1013.876,239.954,-142.041,-24.406,21.386,-41.181
C08573=1013.874,239.706,-142.013,-24.406,21.386,-41.183
C08574=1013.871,239.457,-141.984,-24.406,21.387,-41.184
C08575=1013.869,239.209,-141.956,-24.405,21.387,-41.186
C08576=1013.866,238.961,-141.927,-24.405,21.387,-41.188
C08577=1013.864,238.712,-141.898,-24.405,21.387,-41.190
C08578=1013.861,238.464,-141.870,-24.405,21.388,-41.192
C08579=1013.859,238.215,-141.841,-24.404,21.387,-41.195
C08580=1013.856,237.968,-141.812,-24.404,21.387,-41.197
C08581=1013.853,237.719,-141.784,-24.403,21.388,-41.199
C08582=1013.850,237.470,-141.756,-24.403,21.388,-41.201
C08583=1013.849,237.228,-141.727,-24.403,21.388,-41.203
C08584=1013.846,236.985,-141.700,-24.403,21.388,-41.205
C08585=1013.843,236.742,-141.672,-24.402,21.388,-41.207
C08586=1013.841,236.499,-141.644,-24.402,21.389,-41.209
C08587=1013.838,236.256,-141.616,-24.402,21.389,-41.210
C08588=1013.836,236.013,-141.588,-24.402,21.389,-41.212
C08589=1013.833,235.770,-141.561,-24.401,21.389,-41.214
C08590=1013.831,235.526,-141.533,-24.401,21.390,-41.216
C08591=1013.828,235.279,-141.504,-24.401,21.389,-41.218
C08592=1013.826,235.030,-141.475,-24.401,21.389,-41.219
C08593=1013.823,234.782,-141.447,-24.400,21.389,-41.221
C08594=1013.821,234.534,-141.418,-24.400,21.390,-41.223
C08595=1013.818,234.285,-141.390,-24.400,21.390,-41.225
C08596=1013.816,234.036,-141.362,-24.400,21.390,-41.227
C08597=1013.814,233.789,-141.334,-24.399,21.390,-41.229
C08598=1013.811,233.540,-141.305,-24.399,21.390,-41.231
C08599=1013.808,233.291,-141.277,-24.399,21.391,-41.233
C08600=1013.806,233.044,-141.248,-24.399,21.391,-41.234
C08601=1013.804,232.795,-141.220,-24.398,21.391,-41.236
C08602=1013.801,232.546,-141.191,-24.398,21.390,-41.238
C08603=1013.799,232.298,-141.164,-24.398,21.391,-41.240
C08604=1013.797,232.049,-141.135,-24.397,21.391,-41.242
C08605=1013.794,231.802,-141.107,-24.397,21.391,-41.243
C08606=1013.792,231.553,-141.078,-24.397,21.391,-41.245
C08607=1013.789,231.304,-141.050,-24.397,21.392,-41.247
C08608=1013.787,231.056,-141.022,-24.396,21.392,-41.249
C08609=1013.784,230.808,-140.994,-24.396,21.392,-41.251
C08610=1013.783,230.559,-140.965,-24.396,21.391,-41.252
C08611=1013.780,230.316,-140.938,-24.396,21.392,-41.254
C08612=1013.778,230.073,-140.910,-24.395,21.392,-41.256
C08613=1013.776,229.831,-140.883,-24.395,21.392,-41.258
C08614=1013.773,229.588,-140.855,-24.395,21.392,-41.260
C08615=1013.771,229.345,-140.827,-24.395,21.392,-41.262
C08616=1013.769,229.102,-140.800,-24.394,21.392,-41.263
C08617=1013.767,228.859,-140.772,-24.394,21.392,-41.265
C08618=1013.764,228.616,-140.745,-24.394,21.393,-41.266
C08619=1013.763,228.368,-140.717,-24.394,21.393,-41.267
C08620=1013.760,228.119,-140.689,-24.394,21.393,-41.269
C08621=1013.758,227.871,-140.660,-24.393,21.394,-41.271
C08622=1013.755,227.623,-140.632,-24.393,21.393,-41.273
C08623=1013.753,227.374,-140.604,-24.393,21.393,-41.275
C08624=1013.750,227.126,-140.576,-24.393,21.393,-41.276
C08625=1013.749,226.878,-140.548,-24.392,21.394,-41.278
C08626=1013.746,226.629,-140.519,-24.392,21.394,-41.280
C08627=1013.744,226.381,-140.492,-24.392,21.393,-41.282
C08628=1013.742,226.133,-140.463,-24.391,21.393,-41.284
C08629=1013.740,225.883,-140.436,-24.391,21.394,-41.285
C08630=1013.738,225.636,-140.408,-24.391,21.395,-41.286
C08631=1013.735,225.387,-140.379,-24.391,21.395,-41.288
C08632=1013.733,225.139,-140.351,-24.391,21.394,-41.289
C08633=1013.731,224.891,-140.324,-24.390,21.394,-41.291
C08634=1013.728,224.642,-140.295,-24.390,21.395,-41.293
C08635=1013.726,224.394,-140.267,-24.390,21.395,-41.295
C08636=1013.724,224.145,-140.239,-24.390,21.395,-41.297
C08637=1013.722,223.897,-140.212,-24.389,21.394,-41.298
C08638=1013.720,223.649,-140.183,-24.389,21.395,-41.300
C08639=1013.718,223.406,-140.156,-24.389,21.395,-41.300
C08640=1013.716,223.163,-140.129,-24.389,21.396,-41.302
C08641=1013.714,222.920,-140.102,-24.389,21.396,-41.304
C08642=1013.712,222.677,-140.075,-24.388,21.395,-41.306
C08643=1013.710,222.435,-140.047,-24.388,21.395,-41.308
C08644=1013.708,222.192,-140.020,-24.388,21.396,-41.309
C08645=1013.705,221.949,-139.992,-24.388,21.397,-41.310
C08646=1013.703,221.706,-139.965,-24.388,21.396,-41.311
C08647=1013.701,221.458,-139.938,-24.387,21.396,-41.313
C08648=1013.700,221.209,-139.909,-24.387,21.396,-41.315
C08649=1013.697,220.961,-139.882,-24.387,21.397,-41.317
C08650=1013.695,220.712,-139.854,-24.386,21.396,-41.318
C08651=1013.693,220.464,-139.826,-24.386,21.396,-41.320
C08652=1013.691,220.216,-139.798,-24.386,21.397,-41.321
C08653=1013.689,219.967,-139.770,-24.386,21.397,-41.323
C08654=1013.687,219.718,-139.742,-24.386,21.397,-41.324
C08655=1013.685,219.471,-139.714,-24.385,21.397,-41.326
C08656=1013.683,219.222,-139.687,-24.385,21.397,-41.328
C08657=1013.681,218.974,-139.659,-24.385,21.397,-41.330
C08658=1013.678,218.725,-139.632,-24.385,21.397,-41.330
C08659=1013.677,218.476,-139.603,-24.385,21.397,-41.332
C08660=1013.674,218.229,-139.576,-24.384,21.398,-41.333
C08661=1013.673,217.980,-139.548,-24.384,21.398,-41.335
C08662=1013.671,217.732,-139.520,-24.384,21.397,-41.337
C08663=1013.669,217.482,-139.492,-24.384,21.397,-41.339
C08664=1013.666,217.234,-139.465,-24.384,21.398,-41.339
C08665=1013.665,216.986,-139.437,-24.383,21.399,-41.341
C08666=1013.663,216.738,-139.409,-24.383,21.398,-41.342
C08667=1013.661,216.494,-139.382,-24.383,21.398,-41.344
C08668=1013.659,216.252,-139.355,-24.383,21.398,-41.346
C08669=1013.657,216.010,-139.328,-24.383,21.398,-41.346
C08670=1013.656,215.766,-139.301,-24.382,21.399,-41.348
C08671=1013.654,215.524,-139.274,-24.382,21.399,-41.350
C08672=1013.651,215.281,-139.247,-24.382,21.399,-41.352
C08673=1013.650,215.039,-139.221,-24.382,21.398,-41.353
C08674=1013.648,214.796,-139.193,-24.382,21.399,-41.354
C08675=1013.646,214.548,-139.166,-24.381,21.400,-41.356
C08676=1013.645,214.299,-139.138,-24.381,21.399,-41.357
C08677=1013.643,214.051,-139.111,-24.381,21.399,-41.359
C08678=1013.641,213.803,-139.082,-24.381,21.400,-41.359
C08679=1013.639,213.554,-139.055,-24.381,21.400,-41.361
C08680=1013.638,213.305,-139.028,-24.380,21.400,-41.363
C08681=1013.635,213.057,-139.000,-24.380,21.400,-41.365
C08682=1013.633,212.808,-138.972,-24.380,21.400,-41.366
C08683=1013.631,212.559,-138.945,-24.380,21.400,-41.366
C08684=1013.630,212.311,-138.917,-24.380,21.400,-41.368
C08685=1013.628,212.063,-138.890,-24.379,21.400,-41.370
C08686=1013.626,211.814,-138.862,-24.379,21.400,-41.372
C08687=1013.624,211.566,-138.835,-24.379,21.401,-41.372
C08688=1013.622,211.318,-138.808,-24.379,21.401,-41.374
C08689=1013.621,211.069,-138.780,-24.378,21.400,-41.375
C08690=1013.618,210.821,-138.752,-24.378,21.400,-41.377
C08691=1013.617,210.572,-138.725,-24.378,21.401,-41.378
C08692=1013.615,210.324,-138.698,-24.378,21.401,-41.379
C08693=1013.613,210.075,-138.670,-24.378,21.401,-41.381
C08694=1013.611,209.827,-138.643,-24.377,21.401,-41.383
C08695=1013.610,209.584,-138.616,-24.377,21.401,-41.383
C08696=1013.608,209.342,-138.589,-24.377,21.401,-41.385
C08697=1013.607,209.099,-138.563,-24.377,21.402,-41.387
C08698=1013.604,208.857,-138.535,-24.377,21.401,-41.388
C08699=1013.604,208.614,-138.509,-24.377,21.402,-41.389
C08700=1013.602,208.372,-138.482,-24.376,21.402,-41.391
C08701=1013.600,208.129,-138.455,-24.376,21.401,-41.392
C08702=1013.598,207.886,-138.429,-24.376,21.402,-41.392
C08703=1013.597,207.638,-138.401,-24.376,21.402,-41.394
C08704=1013.595,207.390,-138.374,-24.376,21.402,-41.396
C08705=1013.593,207.141,-138.346,-24.375,21.402,-41.398
C08706=1013.591,206.892,-138.319,-24.375,21.402,-41.398
C08707=1013.590,206.644,-138.292,-24.375,21.402,-41.399
C08708=1013.588,206.395,-138.265,-24.375,21.402,-41.401
C08709=1013.587,206.146,-138.237,-24.375,21.402,-41.401
C08710=1013.585,205.899,-138.210,-24.375,21.403,-41.403
C08711=1013.583,205.650,-138.182,-24.374,21.403,-41.405
C08712=1013.581,205.402,-138.155,-24.374,21.402,-41.407
C08713=1013.580,205.153,-138.128,-24.374,21.403,-41.407
C08714=1013.578,204.904,-138.101,-24.374,21.403,-41.409
C08715=1013.577,204.656,-138.073,-24.373,21.403,-41.410
C08716=1013.575,204.407,-138.046,-24.374,21.404,-41.411
C08717=1013.574,204.159,-138.019,-24.373,21.403,-41.412
C08718=1013.572,203.910,-137.992,-24.373,21.403,-41.414
C08719=1013.571,203.662,-137.965,-24.373,21.404,-41.415
C08720=1013.569,203.413,-137.938,-24.373,21.403,-41.416
C08721=1013.565,202.198,-137.803,-24.425,21.378,-41.051
C08722=1013.565,201.810,-137.760,-24.424,21.378,-41.052
C08723=1013.566,201.461,-137.722,-24.424,21.378,-41.054
C08724=1013.567,201.110,-137.684,-24.424,21.378,-41.058
C08725=1013.568,200.702,-137.640,-24.423,21.379,-41.060
C08726=1013.569,200.475,-137.615,-24.423,21.378,-41.061
C08727=1013.570,200.246,-137.590,-24.423,21.378,-41.063
C08728=1013.570,200.024,-137.565,-24.423,21.378,-41.065
C08729=1013.570,199.811,-137.542,-24.423,21.378,-41.065
C08730=1013.572,199.410,-137.499,-24.422,21.379,-41.069
C08731=1013.573,199.021,-137.456,-24.422,21.379,-41.071
C08732=1013.573,198.623,-137.413,-24.421,21.379,-41.074
C08733=1013.575,198.222,-137.369,-24.421,21.379,-41.076
C08734=1013.576,197.821,-137.326,-24.421,21.380,-41.078
C08735=1013.578,197.419,-137.282,-24.420,21.380,-41.082
C08736=1013.578,197.018,-137.239,-24.420,21.380,-41.084
C08737=1013.580,196.618,-137.196,-24.419,21.380,-41.087
C08738=1013.581,196.216,-137.152,-24.419,21.380,-41.089
C08739=1013.582,195.815,-137.109,-24.419,21.381,-41.091
C08740=1013.583,195.414,-137.065,-24.418,21.380,-41.094
C08741=1013.585,195.013,-137.022,-24.418,21.381,-41.097
C08742=1013.586,194.612,-136.979,-24.418,21.381,-41.100
C08743=1013.587,194.210,-136.935,-24.417,21.381,-41.102
C08744=1013.588,193.810,-136.892,-24.417,21.381,-41.105
C08745=1013.589,193.408,-136.848,-24.417,21.382,-41.108
C08746=1013.591,193.007,-136.805,-24.416,21.382,-41.109
C08747=1013.592,192.606,-136.762,-24.416,21.382,-41.113
C08748=1013.593,192.206,-136.719,-24.415,21.382,-41.115
C08749=1013.595,191.804,-136.675,-24.415,21.382,-41.118
C08750=1013.596,191.402,-136.632,-24.415,21.382,-41.120
C08751=1013.597,191.002,-136.589,-24.414,21.382,-41.124
C08752=1013.598,190.601,-136.546,-24.414,21.383,-41.126
C08753=1013.600,190.200,-136.502,-24.414,21.383,-41.128
C08754=1013.601,189.799,-136.459,-24.413,21.383,-41.131
C08755=1013.602,189.398,-136.416,-24.413,21.383,-41.133
C08756=1013.604,188.997,-136.374,-24.412,21.384,-41.137
C08757=1013.605,188.595,-136.330,-24.412,21.384,-41.139
C08758=1013.607,188.195,-136.287,-24.412,21.384,-41.141
C08759=1013.607,187.794,-136.244,-24.411,21.384,-41.144
C08760=1013.609,187.393,-136.201,-24.411,21.385,-41.146
C08761=1013.611,186.992,-136.158,-24.411,21.384,-41.150
C08762=1013.612,186.591,-136.115,-24.410,21.384,-41.151
C08763=1013.613,186.189,-136.072,-24.410,21.384,-41.155
C08764=1013.615,185.789,-136.029,-24.410,21.385,-41.157
C08765=1013.616,185.388,-135.986,-24.409,21.385,-41.159
C08766=1013.618,184.986,-135.943,-24.409,21.385,-41.162
C08767=1013.619,184.586,-135.900,-24.409,21.386,-41.165
C08768=1013.621,184.185,-135.857,-24.408,21.386,-41.168
C08769=1013.622,183.784,-135.815,-24.408,21.386,-41.170
C08770=1013.624,183.384,-135.772,-24.407,21.386,-41.172
C08771=1013.625,182.982,-135.730,-24.407,21.386,-41.176
C08772=1013.626,182.581,-135.687,-24.407,21.387,-41.177
C08773=1013.628,182.180,-135.643,-24.406,21.386,-41.181
C08774=1013.630,181.779,-135.601,-24.406,21.387,-41.183
C08775=1013.631,181.379,-135.558,-24.405,21.387,-41.186
C08776=1013.633,180.978,-135.516,-24.405,21.387,-41.188
C08777=1013.634,180.577,-135.473,-24.405,21.387,-41.190
C08778=1013.636,180.176,-135.430,-24.404,21.388,-41.194
C08779=1013.637,179.776,-135.388,-24.404,21.388,-41.196
C08780=1013.639,179.374,-135.345,-24.403,21.388,-41.199
C08781=1013.640,178.974,-135.302,-24.403,21.388,-41.201
C08782=1013.642,178.573,-135.260,-24.403,21.388,-41.205
C08783=1013.643,178.172,-135.217,-24.402,21.388,-41.207
C08784=1013.645,177.771,-135.175,-24.402,21.389,-41.209
C08785=1013.646,177.371,-135.132,-24.402,21.389,-41.212
C08786=1013.648,176.970,-135.090,-24.401,21.389,-41.214
C08787=1013.649,176.569,-135.047,-24.401,21.389,-41.218
C08788=1013.651,176.169,-135.005,-24.401,21.389,-41.219
C08789=1013.653,175.767,-134.963,-24.400,21.390,-41.223
C08790=1013.654,175.367,-134.920,-24.400,21.390,-41.225
C08791=1013.656,174.966,-134.878,-24.400,21.390,-41.227
C08792=1013.657,174.565,-134.835,-24.399,21.390,-41.231
C08793=1013.660,174.165,-134.793,-24.399,21.391,-41.233
C08794=1013.661,173.764,-134.751,-24.398,21.390,-41.236
C08795=1013.662,173.364,-134.708,-24.398,21.390,-41.238
C08796=1013.664,172.963,-134.666,-24.397,21.391,-41.242
C08797=1013.666,172.563,-134.623,-24.397,21.391,-41.243
C08798=1013.667,172.162,-134.581,-24.397,21.391,-41.247
C08799=1013.670,171.761,-134.539,-24.396,21.392,-41.249
C08800=1013.670,171.361,-134.497,-24.396,21.392,-41.251
C08801=1013.672,170.961,-134.455,-24.396,21.392,-41.254
C08802=1013.674,170.559,-134.413,-24.395,21.392,-41.256
C08803=1013.676,170.160,-134.370,-24.395,21.392,-41.260
C08804=1013.678,169.758,-134.328,-24.395,21.392,-41.262
C08805=1013.679,169.358,-134.287,-24.394,21.392,-41.265
C08806=1013.681,168.958,-134.244,-24.394,21.393,-41.267
C08807=1013.683,168.557,-134.202,-24.393,21.393,-41.271
C08808=1013.684,168.157,-134.160,-24.393,21.393,-41.273
C08809=1013.686,167.756,-134.118,-24.393,21.394,-41.275
C08810=1013.688,167.356,-134.076,-24.392,21.394,-41.278
C08811=1013.690,166.955,-134.034,-24.392,21.394,-41.280
C08812=1013.691,166.555,-133.992,-24.391,21.393,-41.284
C08813=1013.693,166.155,-133.950,-24.391,21.395,-41.286
C08814=1013.694,165.755,-133.908,-24.391,21.394,-41.289
C08815=1013.696,165.354,-133.866,-24.390,21.394,-41.291
C08816=1013.698,164.954,-133.824,-24.390,21.395,-41.295
C08817=1013.699,164.554,-133.782,-24.390,21.395,-41.297
C08818=1013.701,164.153,-133.740,-24.389,21.395,-41.300
C08819=1013.703,163.767,-133.700,-24.389,21.395,-41.302
C08820=1013.704,163.578,-133.680,-24.389,21.395,-41.304
C08821=1013.705,163.166,-133.637,-24.388,21.396,-41.306
C08822=1013.707,162.930,-133.613,-24.388,21.395,-41.308
C08823=1013.708,162.676,-133.585,-24.388,21.396,-41.309
C08824=1013.709,162.414,-133.559,-24.388,21.396,-41.311
C08825=1013.710,162.145,-133.531,-24.387,21.396,-41.313
C08826=1013.712,161.873,-133.502,-24.387,21.396,-41.315
C08827=1013.712,161.604,-133.475,-24.387,21.397,-41.317
C08828=1013.714,161.342,-133.447,-24.387,21.397,-41.319
C08829=1013.715,161.091,-133.420,-24.386,21.396,-41.320
C08830=1013.716,160.853,-133.396,-24.386,21.396,-41.322
C08831=1013.717,160.629,-133.372,-24.386,21.397,-41.324
C08832=1013.718,160.415,-133.351,-24.386,21.397,-41.325
C08833=1013.720,160.010,-133.308,-24.385,21.397,-41.328
C08834=1013.725,159.614,-133.269,-24.385,21.397,-41.330
C08835=1013.735,159.214,-133.233,-24.384,21.398,-41.333
C08836=1013.745,158.814,-133.195,-24.384,21.398,-41.335
C08837=1013.754,158.413,-133.160,-24.384,21.397,-41.339
C08838=1013.764,158.011,-133.122,-24.383,21.399,-41.341
C08839=1013.773,157.609,-133.085,-24.383,21.398,-41.344
C08840=1013.783,157.206,-133.047,-24.383,21.398,-41.346
C08841=1013.792,156.801,-133.010,-24.382,21.399,-41.350
C08842=1013.802,156.396,-132.973,-24.382,21.399,-41.352
C08843=1013.811,155.991,-132.935,-24.381,21.399,-41.355
C08844=1013.821,155.584,-132.898,-24.381,21.400,-41.358
C08845=1013.830,155.177,-132.861,-24.381,21.399,-41.361
C08846=1013.840,154.768,-132.823,-24.380,21.400,-41.363
C08847=1013.848,154.359,-132.785,-24.380,21.400,-41.366
C08848=1013.858,153.949,-132.748,-24.380,21.400,-41.368
C08849=1013.867,153.539,-132.710,-24.379,21.401,-41.372
C08850=1013.876,153.128,-132.671,-24.378,21.400,-41.375
C08851=1013.886,152.717,-132.633,-24.378,21.400,-41.377
C08852=1013.895,152.304,-132.596,-24.378,21.401,-41.381
C08853=1013.904,151.892,-132.557,-24.377,21.401,-41.383
C08854=1013.914,151.480,-132.519,-24.377,21.402,-41.387
C08855=1013.923,151.066,-132.481,-24.377,21.402,-41.389
C08856=1013.931,150.653,-132.443,-24.376,21.401,-41.392
C08857=1013.941,150.239,-132.404,-24.376,21.402,-41.394
C08858=1013.950,149.825,-132.366,-24.375,21.402,-41.398
C08859=1013.959,149.411,-132.328,-24.375,21.402,-41.401
C08860=1013.968,148.998,-132.290,-24.375,21.403,-41.403
C08861=1013.976,148.583,-132.251,-24.374,21.403,-41.407
C08862=1013.985,148.170,-132.213,-24.374,21.403,-41.409
C08863=1013.994,147.756,-132.175,-24.373,21.403,-41.412
C08864=1014.003,147.343,-132.136,-24.373,21.403,-41.416
C08865=1014.012,146.929,-132.099,-24.372,21.404,-41.418
C08866=1014.020,146.516,-132.060,-24.372,21.404,-41.422
C08867=1014.029,146.103,-132.022,-24.372,21.404,-41.424
C08868=1014.037,145.690,-131.983,-24.371,21.405,-41.427
C08869=1014.046,145.278,-131.945,-24.371,21.404,-41.431
C08870=1014.055,144.866,-131.907,-24.370,21.405,-41.432
C08871=1014.063,144.455,-131.869,-24.370,21.405,-41.436
C08872=1014.072,144.044,-131.831,-24.370,21.405,-41.438
C08873=1014.080,143.634,-131.793,-24.369,21.406,-41.442
C08874=1014.089,143.224,-131.755,-24.369,21.405,-41.445
C08875=1014.097,142.816,-131.717,-24.368,21.406,-41.448
C08876=1014.105,142.408,-131.680,-24.368,21.406,-41.451
C08877=1014.113,142.000,-131.642,-24.368,21.406,-41.453
C08878=1014.121,141.594,-131.604,-24.367,21.407,-41.457
C08879=1014.129,141.189,-131.566,-24.366,21.406,-41.460
C08880=1014.138,140.786,-131.529,-24.366,21.407,-41.462
C08881=1014.146,140.368,-131.490,-24.366,21.408,-41.466
C08882=1014.151,140.132,-131.468,-24.366,21.408,-41.468
C08883=1014.155,139.874,-131.445,-24.365,21.408,-41.470
C08884=1014.161,139.597,-131.418,-24.365,21.408,-41.471
C08885=1014.166,139.309,-131.392,-24.365,21.408,-41.473
C08886=1014.172,139.022,-131.365,-24.364,21.408,-41.475
C08887=1014.178,138.744,-131.339,-24.364,21.407,-41.476
C08888=1014.182,138.484,-131.315,-24.364,21.408,-41.478
C08889=1014.187,138.247,-131.294,-24.364,21.408,-41.480
C08890=1014.192,138.030,-131.273,-24.363,21.408,-41.482
C08891=1014.195,137.825,-131.254,-24.363,21.408,-41.484
C08892=1014.203,137.424,-131.218,-24.363,21.408,-41.486
C08893=1014.210,137.054,-131.182,-24.363,21.410,-41.488
C08894=1014.216,136.717,-131.152,-24.362,21.409,-41.491
C08895=1014.223,136.401,-131.122,-24.361,21.409,-41.495
C08896=1014.228,136.084,-131.093,-24.361,21.410,-41.497
C08897=1014.235,135.744,-131.061,-24.361,21.409,-41.500
C08898=1014.242,135.373,-131.027,-24.360,21.410,-41.502
C08899=1014.249,134.978,-130.990,-24.360,21.411,-41.505
C08900=1014.257,134.580,-130.953,-24.360,21.410,-41.508
C08901=1014.265,134.181,-130.916,-24.359,21.411,-41.510
C08902=1014.272,133.782,-130.879,-24.359,21.411,-41.514
C08903=1014.279,133.383,-130.842,-24.358,21.411,-41.517
C08904=1014.287,132.984,-130.805,-24.358,21.412,-41.519
C08905=1014.294,132.586,-130.768,-24.358,21.411,-41.523
C08906=1014.301,132.188,-130.730,-24.357,21.412,-41.525
C08907=1014.308,131.790,-130.694,-24.357,21.412,-41.528
C08908=1014.315,131.391,-130.657,-24.356,21.412,-41.532
C08909=1014.323,130.992,-130.620,-24.356,21.413,-41.534
C08910=1014.330,130.593,-130.583,-24.356,21.413,-41.538
C08911=1014.337,130.195,-130.546,-24.355,21.413,-41.541
C08912=1014.344,129.797,-130.509,-24.355,21.413,-41.543
C08913=1014.351,129.398,-130.472,-24.354,21.413,-41.547
C08914=1014.358,128.999,-130.435,-24.354,21.413,-41.550
C08915=1014.365,128.601,-130.398,-24.354,21.414,-41.552
C08916=1014.372,128.203,-130.361,-24.353,21.414,-41.555
C08917=1014.379,127.804,-130.324,-24.353,21.415,-41.558
C08918=1014.386,127.405,-130.287,-24.352,21.414,-41.561
C08919=1014.393,127.007,-130.250,-24.352,21.415,-41.565
C08920=1014.400,126.609,-130.213,-24.351,21.415,-41.567
C08921=1014.407,126.211,-130.175,-24.351,21.415,-41.571
C08922=1014.414,125.812,-130.139,-24.350,21.415,-41.574
C08923=1014.421,125.413,-130.102,-24.350,21.416,-41.576
C08924=1014.427,125.016,-130.065,-24.350,21.416,-41.580
C08925=1014.434,124.617,-130.028,-24.349,21.416,-41.583
C08926=1014.441,124.218,-129.991,-24.349,21.416,-41.585
C08927=1014.447,123.820,-129.953,-24.348,21.417,-41.589
C08928=1014.454,123.421,-129.917,-24.348,21.416,-41.592
C08929=1014.460,123.023,-129.880,-24.348,21.418,-41.595
C08930=1014.468,122.625,-129.843,-24.347,21.417,-41.598
C08931=1014.474,122.227,-129.805,-24.347,21.418,-41.602
C08932=1014.480,121.827,-129.769,-24.346,21.417,-41.605
C08933=1014.487,121.429,-129.732,-24.346,21.418,-41.607
C08934=1014.493,121.031,-129.695,-24.345,21.418,-41.611
C08935=1014.500,120.632,-129.658,-24.345,21.418,-41.614
C08936=1014.507,120.234,-129.621,-24.345,21.419,-41.617
C08937=1014.514,119.836,-129.584,-24.344,21.419,-41.620
C08938=1014.520,119.437,-129.548,-24.343,21.419,-41.624
C08939=1014.528,119.039,-129.511,-24.343,21.420,-41.626
C08940=1014.535,118.640,-129.474,-24.343,21.420,-41.629
C08941=1014.541,118.242,-129.438,-24.342,21.420,-41.633
C08942=1014.548,117.843,-129.401,-24.342,21.420,-41.637
C08943=1014.555,117.446,-129.364,-24.341,21.420,-41.638
C08944=1014.562,117.047,-129.328,-24.341,21.421,-41.642
C08945=1014.569,116.649,-129.291,-24.340,21.420,-41.646
C08946=1014.575,116.250,-129.255,-24.340,21.421,-41.649
C08947=1014.582,115.852,-129.218,-24.340,21.422,-41.652
C08948=1014.588,115.454,-129.181,-24.339,21.422,-41.655
C08949=1014.595,115.055,-129.144,-24.339,21.422,-41.659
C08950=1014.601,114.656,-129.107,-24.338,21.422,-41.662
C08951=1014.608,114.258,-129.071,-24.338,21.423,-41.664
C08952=1014.615,113.859,-129.034,-24.337,21.422,-41.668
C08953=1014.621,113.462,-128.998,-24.337,21.423,-41.671
C08954=1014.628,113.063,-128.961,-24.336,21.423,-41.675
C08955=1014.634,112.665,-128.925,-24.336,21.423,-41.677
C08956=1014.641,112.266,-128.888,-24.335,21.424,-41.681
C08957=1014.647,111.868,-128.851,-24.335,21.423,-41.684
C08958=1014.653,111.469,-128.814,-24.334,21.424,-41.688
